(* IEC 61131-3 sources: PortalRobot/Portal_robot/Device/application/FB (part 2) *)

(* ---- FB_CELL_SAFETY.st ---- *)
FUNCTION_BLOCK FB_CELL_SAFETY
VAR_INPUT
	axDoorLockClosedInput : ARRAY [1..4] OF BOOL;
	axDoorUnlockButtonInput : ARRAY [1..4] OF BOOL;
	axMagazineMechanismBusy : ARRAY [1..2] OF BOOL; // Только новый механизм, включая фактическое движение оси
	axEmergencyStopButtonStationInput : ARRAY [1..4] OF BOOL;
	axEmergencyStopCabinetInput : ARRAY [1..2] OF BOOL;
	xEmergencyStopMpgInput : BOOL;
	xPhaseRelayOkInput    : BOOL;
	xPressureRelayOkInput : BOOL;
	xSafetyRelayOkInput   : BOOL;
	xCellStartButtonInput : BOOL;
	xCellStopButtonInput  : BOOL;
	xCellResetButtonInput : BOOL;
	xMpgAxisXInput : BOOL;
	xMpgAxisYInput : BOOL;
	xMpgAxisZInput : BOOL;
	xMpgMultiplier1Input : BOOL;
	xMpgMultiplier10Input : BOOL;
	xMpgMultiplier100Input : BOOL;
	xSafetyRelayReset : BOOL; // Импульс отдельного сброса реле безопасности
	astMagazineStatus : ARRAY [1..2] OF ST_MAGAZINE_STATUS;
	FaultRequest : ST_CELL_SAFETY_FAULT_REQUEST;
END_VAR
VAR_OUTPUT
	Status : ST_CELL_SAFETY_STATUS;
	Error  : ST_CELL_SAFETY_ERRORS;
	Diag   : ST_CELL_SAFETY_DIAG;
	FaultStatus : ST_FAULT_INJECTION_STATUS;
	astButtonStationIoStatus : ARRAY [1..4] OF ST_BUTTON_STATION_IO_STATUS;
	stFrontControlCabinetIoStatus : ST_CONTROL_CABINET_IO_STATUS;
	stRearControlCabinetIoStatus : ST_CONTROL_CABINET_IO_STATUS;
	stMpgIoStatus : ST_MPG_IO_STATUS;
	astEnclosureDoorStatus : ARRAY [1..4] OF ST_ENCLOSURE_DOOR_STATUS;
	axDoorUnlockOutput : ARRAY [1..4] OF BOOL;
	axDoorButtonLampOutput : ARRAY [1..4] OF BOOL;
	xSafetyRelayResetOutput : BOOL;
	xCellEnablePulse : BOOL;
	xCellDisablePulse : BOOL;
	xCellResetPulse : BOOL;
END_VAR
VAR
	fbFaultInjector : FB_CELL_SAFETY_FAULT_INJECTOR;
	axEmergencyStopStation : ARRAY [1..4] OF BOOL;
	axEmergencyStopCabinet : ARRAY [1..2] OF BOOL;
	axDoorLocked : ARRAY [1..4] OF BOOL;
	axDoorUnlockDemand : ARRAY [1..4] OF BOOL;
	axDoorSeenUnlocked : ARRAY [1..4] OF BOOL;
	artDoorButton : ARRAY [1..4] OF R_TRIG;
	rtSafetyRelayReset : R_TRIG;
	tpSafetyRelayReset : TP;
	rtCellStart : R_TRIG;
	rtCellStop : R_TRIG;
	rtCellReset : R_TRIG;
	xEmergencyStopMpg : BOOL;
	xPhaseRelayOk : BOOL;
	xPressureRelayOk : BOOL;
	xSafetyRelayOk : BOOL;
	dwLiveFaultMask : DWORD;
	uiDoor : UINT;
	uiMagazine : UINT;
END_VAR
VAR CONSTANT
	ERR_ESTOP_STATION_1 : DWORD := DWORD#16#0000_0001;
	ERR_ESTOP_STATION_2 : DWORD := DWORD#16#0000_0002;
	ERR_ESTOP_STATION_3 : DWORD := DWORD#16#0000_0004;
	ERR_ESTOP_STATION_4 : DWORD := DWORD#16#0000_0008;
	ERR_ESTOP_CABINET_FRONT : DWORD := DWORD#16#0000_0010;
	ERR_ESTOP_CABINET_REAR  : DWORD := DWORD#16#0000_0020;
	ERR_ESTOP_MPG      : DWORD := DWORD#16#0000_0040;
	ERR_PHASE_RELAY    : DWORD := DWORD#16#0000_0080;
	ERR_PRESSURE_RELAY : DWORD := DWORD#16#0000_0100;
	ERR_SAFETY_RELAY   : DWORD := DWORD#16#0000_0200;
	ERR_DOOR_1_UNLOCKED : DWORD := DWORD#16#0000_0400;
	ERR_DOOR_2_UNLOCKED : DWORD := DWORD#16#0000_0800;
	ERR_DOOR_3_UNLOCKED : DWORD := DWORD#16#0000_1000;
	ERR_DOOR_4_UNLOCKED : DWORD := DWORD#16#0000_2000;
	WRN_SAFETY_RESET_REJECTED : UINT := UINT#1;
	WRN_DOOR_1_UNLOCK_REJECTED : UINT := UINT#2;
END_VAR

// --- BEGIN IMPLEMENTATION ---

fbFaultInjector(Request := FaultRequest);
FaultStatus := fbFaultInjector.Status;

FOR uiDoor := UINT#1 TO UINT#4 DO
	axEmergencyStopStation[uiDoor] := axEmergencyStopButtonStationInput[uiDoor]
		OR fbFaultInjector.axEmergencyStopStation[uiDoor];
	axDoorLocked[uiDoor] := axDoorLockClosedInput[uiDoor]
		AND NOT fbFaultInjector.axDoorUnlocked[uiDoor];
	artDoorButton[uiDoor](CLK := axDoorUnlockButtonInput[uiDoor]);

	IF uiDoor <= UINT#2 THEN
		uiMagazine := UINT#1;
	ELSE
		uiMagazine := UINT#2;
	END_IF;
	astEnclosureDoorStatus[uiDoor].xUnlockAllowed := NOT astMagazineStatus[uiMagazine].xEnabled AND NOT axMagazineMechanismBusy[uiMagazine];
	axDoorButtonLampOutput[uiDoor] := astEnclosureDoorStatus[uiDoor].xUnlockAllowed;

	IF artDoorButton[uiDoor].Q THEN
		IF astEnclosureDoorStatus[uiDoor].xUnlockAllowed THEN
			axDoorUnlockDemand[uiDoor] := TRUE;
			axDoorSeenUnlocked[uiDoor] := FALSE;
		ELSE
			RaiseWarning(uiCode := WRN_DOOR_1_UNLOCK_REJECTED + uiDoor - UINT#1);
		END_IF;
	END_IF;

	// Команда держится до фактического цикла «замок открылся -> снова закрылся».
	// Если магазин включили поверх открытого доступа, выход снимается немедленно.
	IF NOT astEnclosureDoorStatus[uiDoor].xUnlockAllowed THEN
		axDoorUnlockDemand[uiDoor] := FALSE;
		axDoorSeenUnlocked[uiDoor] := FALSE;
	ELSIF axDoorUnlockDemand[uiDoor] THEN
		IF NOT axDoorLocked[uiDoor] THEN
			axDoorSeenUnlocked[uiDoor] := TRUE;
		ELSIF axDoorSeenUnlocked[uiDoor] THEN
			axDoorUnlockDemand[uiDoor] := FALSE;
			axDoorSeenUnlocked[uiDoor] := FALSE;
		END_IF;
	END_IF;

	axDoorUnlockOutput[uiDoor] := axDoorUnlockDemand[uiDoor];
	astEnclosureDoorStatus[uiDoor].xLocked := axDoorLocked[uiDoor];
	astEnclosureDoorStatus[uiDoor].xUnlockOutput := axDoorUnlockOutput[uiDoor];
	astButtonStationIoStatus[uiDoor].xEmergencyStopPressed := axEmergencyStopStation[uiDoor];
	astButtonStationIoStatus[uiDoor].xButtonPressed := axDoorUnlockButtonInput[uiDoor];
	astButtonStationIoStatus[uiDoor].xButtonLightOn := axDoorButtonLampOutput[uiDoor];
	Status.axEmergencyStopReleased[uiDoor] := NOT axEmergencyStopStation[uiDoor];
	Status.axDoorReady[uiDoor] := astEnclosureDoorStatus[uiDoor].xUnlockAllowed OR axDoorLocked[uiDoor];
	Status.axButtonStationPressed[uiDoor] := astButtonStationIoStatus[uiDoor].xButtonPressed;
	Status.axButtonStationLightOn[uiDoor] := astButtonStationIoStatus[uiDoor].xButtonLightOn;
END_FOR;

FOR uiDoor := UINT#1 TO UINT#2 DO
	axEmergencyStopCabinet[uiDoor] := axEmergencyStopCabinetInput[uiDoor]
		OR fbFaultInjector.axEmergencyStopCabinet[uiDoor];
	Status.axEmergencyStopReleased[uiDoor + UINT#4] := NOT axEmergencyStopCabinet[uiDoor];
END_FOR;
xEmergencyStopMpg := xEmergencyStopMpgInput OR fbFaultInjector.xEmergencyStopMpg;
Status.axEmergencyStopReleased[7] := NOT xEmergencyStopMpg;

xPhaseRelayOk := xPhaseRelayOkInput AND NOT fbFaultInjector.xPhaseRelayFault;
xPressureRelayOk := xPressureRelayOkInput AND NOT fbFaultInjector.xPressureRelayFault;
xSafetyRelayOk := xSafetyRelayOkInput AND NOT fbFaultInjector.xSafetyRelayFault;

rtSafetyRelayReset(CLK := xSafetyRelayReset);
Status.xSafetyRelayResetAllowed := NOT xSafetyRelayOk AND NOT tpSafetyRelayReset.Q;
IF rtSafetyRelayReset.Q AND NOT Status.xSafetyRelayResetAllowed THEN
	RaiseWarning(uiCode := WRN_SAFETY_RESET_REJECTED);
END_IF;
tpSafetyRelayReset(
	IN := rtSafetyRelayReset.Q AND Status.xSafetyRelayResetAllowed,
	PT := T#1S
);
// Разрешение проверяется на фронте команды; после запуска выдаём полный импульс 1 с.
xSafetyRelayResetOutput := tpSafetyRelayReset.Q;
Status.xSafetyRelayResetActive := xSafetyRelayResetOutput;

rtCellStart(CLK := xCellStartButtonInput);
rtCellStop(CLK := xCellStopButtonInput);
rtCellReset(CLK := xCellResetButtonInput);
xCellEnablePulse := rtCellStart.Q;
xCellDisablePulse := rtCellStop.Q;
xCellResetPulse := rtCellReset.Q;

stFrontControlCabinetIoStatus.xEmergencyStopPressed := axEmergencyStopCabinet[1];
stFrontControlCabinetIoStatus.xStartPressed := xCellStartButtonInput;
stFrontControlCabinetIoStatus.xStopPressed := xCellStopButtonInput;
stFrontControlCabinetIoStatus.xResetPressed := xCellResetButtonInput;
stRearControlCabinetIoStatus.xEmergencyStopPressed := axEmergencyStopCabinet[2];
stRearControlCabinetIoStatus.xStartPressed := FALSE;
stRearControlCabinetIoStatus.xStopPressed := FALSE;
stRearControlCabinetIoStatus.xResetPressed := FALSE;
stMpgIoStatus.xEmergencyStopPressed := xEmergencyStopMpg;
stMpgIoStatus.xAxisX := xMpgAxisXInput;
stMpgIoStatus.xAxisY := xMpgAxisYInput;
stMpgIoStatus.xAxisZ := xMpgAxisZInput;
stMpgIoStatus.xMultiplier1 := xMpgMultiplier1Input;
stMpgIoStatus.xMultiplier10 := xMpgMultiplier10Input;
stMpgIoStatus.xMultiplier100 := xMpgMultiplier100Input;

dwLiveFaultMask := DWORD#0;
IF axEmergencyStopStation[1] THEN dwLiveFaultMask := dwLiveFaultMask OR ERR_ESTOP_STATION_1; END_IF;
IF axEmergencyStopStation[2] THEN dwLiveFaultMask := dwLiveFaultMask OR ERR_ESTOP_STATION_2; END_IF;
IF axEmergencyStopStation[3] THEN dwLiveFaultMask := dwLiveFaultMask OR ERR_ESTOP_STATION_3; END_IF;
IF axEmergencyStopStation[4] THEN dwLiveFaultMask := dwLiveFaultMask OR ERR_ESTOP_STATION_4; END_IF;
IF axEmergencyStopCabinet[1] THEN dwLiveFaultMask := dwLiveFaultMask OR ERR_ESTOP_CABINET_FRONT; END_IF;
IF axEmergencyStopCabinet[2] THEN dwLiveFaultMask := dwLiveFaultMask OR ERR_ESTOP_CABINET_REAR; END_IF;
IF xEmergencyStopMpg THEN dwLiveFaultMask := dwLiveFaultMask OR ERR_ESTOP_MPG; END_IF;
IF NOT xPhaseRelayOk THEN dwLiveFaultMask := dwLiveFaultMask OR ERR_PHASE_RELAY; END_IF;
IF NOT xPressureRelayOk THEN dwLiveFaultMask := dwLiveFaultMask OR ERR_PRESSURE_RELAY; END_IF;
IF NOT xSafetyRelayOk THEN dwLiveFaultMask := dwLiveFaultMask OR ERR_SAFETY_RELAY; END_IF;
IF (astMagazineStatus[1].xEnabled OR axMagazineMechanismBusy[1]) AND NOT axDoorLocked[1] THEN dwLiveFaultMask := dwLiveFaultMask OR ERR_DOOR_1_UNLOCKED; END_IF;
IF (astMagazineStatus[1].xEnabled OR axMagazineMechanismBusy[1]) AND NOT axDoorLocked[2] THEN dwLiveFaultMask := dwLiveFaultMask OR ERR_DOOR_2_UNLOCKED; END_IF;
IF (astMagazineStatus[2].xEnabled OR axMagazineMechanismBusy[2]) AND NOT axDoorLocked[3] THEN dwLiveFaultMask := dwLiveFaultMask OR ERR_DOOR_3_UNLOCKED; END_IF;
IF (astMagazineStatus[2].xEnabled OR axMagazineMechanismBusy[2]) AND NOT axDoorLocked[4] THEN dwLiveFaultMask := dwLiveFaultMask OR ERR_DOOR_4_UNLOCKED; END_IF;

Error.dwErrorActive := dwLiveFaultMask;
Error.dwAlarmActive := dwLiveFaultMask;
IF dwLiveFaultMask <> DWORD#0 THEN
	Error.dwErrorLast := dwLiveFaultMask;
END_IF;
Status.xPhaseRelayOk := xPhaseRelayOk;
Status.xPressureRelayOk := xPressureRelayOk;
Status.xSafetyRelayOk := xSafetyRelayOk;
Status.xGlobalError := dwLiveFaultMask <> DWORD#0;
Status.xReady := NOT Status.xGlobalError;

(* ---- FB_GRIPPER_SIMULATION.st ---- *)
FUNCTION_BLOCK FB_GRIPPER_SIMULATION
VAR_INPUT
	Command : ST_GRIPPER_COMMAND; // Команда управления захватом

    xSimGripper1Fault : BOOL; // Имитация неисправности первого захвата
    xSimGripper2Fault : BOOL; // Имитация неисправности второго захвата
    xSimRotationFault : BOOL; // Имитация неисправности поворота
    xSimGlobalFault   : BOOL; // Имитация общей неисправности захвата

    tGripperTime : TIME := T#500MS; // Время открытия или закрытия захвата
    tRotateTime  : TIME := T#700MS; // Время поворота захвата
END_VAR
VAR_OUTPUT
	Status : ST_GRIPPER_STATUS; // Рабочие статусы захвата
	Diag   : ST_GRIPPER_DIAG; // Состояние автомата и активное действие
	Error  : ST_GRIPPER_ERRORS; // Активные и последние ошибки
END_VAR
VAR
	eState        : E_GRIPPER_STATE := E_GRIPPER_STATE.IDLE; // Текущее состояние автомата захвата
    eActiveAction : E_ROBOT_ACTION := E_ROBOT_ACTION.NONE; // Выполняемое действие захвата

    tonAction      : TON; // Таймер выполнения действия
    xActionFault   : BOOL; // Неисправность, относящаяся к текущему действию
	xActionValid   : BOOL; // Получено допустимое действие захвата
	xActionRequired: BOOL; // Для действия требуется физическое переключение
    tActionTime    : TIME; // Нормативное время текущего действия
    xInitialized   : BOOL; // Начальные состояния установлены
END_VAR
VAR CONSTANT
	ERR_GRIPPER_1   : DWORD := DWORD#16#0000_0001; // Ошибка первого захвата
    ERR_GRIPPER_2   : DWORD := DWORD#16#0000_0002; // Ошибка второго захвата
    ERR_GRIP_ROTATE : DWORD := DWORD#16#0000_0004; // Ошибка механизма поворота
    ERR_GRIP_ACTION : DWORD := DWORD#16#0000_0008; // Недопустимое действие захвата
    ERR_GRIP_GLOBAL : DWORD := DWORD#16#0000_0010; // Общая ошибка захвата
END_VAR

// --- BEGIN IMPLEMENTATION ---

IF NOT xInitialized THEN
    Status.xGripper1Open := TRUE;
    Status.xGripper1Closed := FALSE;

    Status.xGripper2Open := TRUE;
    Status.xGripper2Closed := FALSE;

    Status.xRotatedToBlank := TRUE;
    Status.xRotatedToDetail := FALSE;

    xInitialized := TRUE;
END_IF;

xActionFault := FALSE;
tActionTime := tGripperTime;

CASE eActiveAction OF

    E_ROBOT_ACTION.UNCLAMP_1,
    E_ROBOT_ACTION.CLAMP_1:
        xActionFault := xSimGripper1Fault;

    E_ROBOT_ACTION.UNCLAMP_2,
    E_ROBOT_ACTION.CLAMP_2:
        xActionFault := xSimGripper2Fault;

    E_ROBOT_ACTION.ROTATE_TO_BLANK,
    E_ROBOT_ACTION.ROTATE_TO_DETAIL:
        xActionFault := xSimRotationFault;
        tActionTime := tRotateTime;

END_CASE;

tonAction(
    IN := (eState = E_GRIPPER_STATE.EXECUTE)
          AND NOT xActionFault
          AND NOT xSimGlobalFault,
    PT := tActionTime
);

CASE eState OF

    E_GRIPPER_STATE.IDLE:

        Status.xBusy := FALSE;
        Status.xDone := FALSE;
        Status.xError := FALSE;

        IF Command.xExecute THEN
            eActiveAction := Command.eAction;
			xActionValid := TRUE;
			xActionRequired := TRUE;

            CASE Command.eAction OF

				E_ROBOT_ACTION.UNCLAMP_1:
					xActionRequired := NOT Status.xGripper1Open;

				E_ROBOT_ACTION.CLAMP_1:
					xActionRequired := NOT Status.xGripper1Closed;

				E_ROBOT_ACTION.UNCLAMP_2:
					xActionRequired := NOT Status.xGripper2Open;

				E_ROBOT_ACTION.CLAMP_2:
					xActionRequired := NOT Status.xGripper2Closed;

				E_ROBOT_ACTION.ROTATE_TO_BLANK:
					xActionRequired := NOT Status.xRotatedToBlank;

				E_ROBOT_ACTION.ROTATE_TO_DETAIL:
					xActionRequired := NOT Status.xRotatedToDetail;

            ELSE
				xActionValid := FALSE;
                Error.dwErrorActive := Error.dwErrorActive OR ERR_GRIP_ACTION;
                eState := E_GRIPPER_STATE.ERROR;
            END_CASE;

			IF xActionValid THEN
				IF xActionRequired THEN
					eState := E_GRIPPER_STATE.EXECUTE;
				ELSE
					eState := E_GRIPPER_STATE.DONE;
				END_IF;
			END_IF;
        END_IF;

    E_GRIPPER_STATE.EXECUTE:

        Status.xBusy := TRUE;
        Status.xDone := FALSE;

        IF xSimGlobalFault THEN
            Error.dwErrorActive := Error.dwErrorActive OR ERR_GRIP_GLOBAL;
            eState := E_GRIPPER_STATE.ERROR;

        ELSIF xActionFault THEN

            CASE eActiveAction OF

                E_ROBOT_ACTION.UNCLAMP_1,
                E_ROBOT_ACTION.CLAMP_1:
                    Error.dwErrorActive := Error.dwErrorActive OR ERR_GRIPPER_1;

                E_ROBOT_ACTION.UNCLAMP_2,
                E_ROBOT_ACTION.CLAMP_2:
                    Error.dwErrorActive := Error.dwErrorActive OR ERR_GRIPPER_2;

                E_ROBOT_ACTION.ROTATE_TO_BLANK,
                E_ROBOT_ACTION.ROTATE_TO_DETAIL:
                    Error.dwErrorActive := Error.dwErrorActive OR ERR_GRIP_ROTATE;

            END_CASE;

            eState := E_GRIPPER_STATE.ERROR;

        ELSIF tonAction.Q THEN

            CASE eActiveAction OF

                E_ROBOT_ACTION.UNCLAMP_1:
                    Status.xGripper1Open := TRUE;
                    Status.xGripper1Closed := FALSE;

                E_ROBOT_ACTION.CLAMP_1:
                    Status.xGripper1Open := FALSE;
                    Status.xGripper1Closed := TRUE;

                E_ROBOT_ACTION.UNCLAMP_2:
                    Status.xGripper2Open := TRUE;
                    Status.xGripper2Closed := FALSE;

                E_ROBOT_ACTION.CLAMP_2:
                    Status.xGripper2Open := FALSE;
                    Status.xGripper2Closed := TRUE;

                E_ROBOT_ACTION.ROTATE_TO_BLANK:
                    Status.xRotatedToBlank := TRUE;
                    Status.xRotatedToDetail := FALSE;

                E_ROBOT_ACTION.ROTATE_TO_DETAIL:
                    Status.xRotatedToBlank := FALSE;
                    Status.xRotatedToDetail := TRUE;

            END_CASE;

            eState := E_GRIPPER_STATE.DONE;
        END_IF;

    E_GRIPPER_STATE.DONE:

        Status.xBusy := FALSE;
        Status.xDone := TRUE;

        IF NOT Command.xExecute THEN
            Status.xDone := FALSE;
            eActiveAction := E_ROBOT_ACTION.NONE;
            eState := E_GRIPPER_STATE.IDLE;
        END_IF;

    E_GRIPPER_STATE.ERROR:

        Status.xBusy := FALSE;
        Status.xDone := FALSE;
        Status.xError := TRUE;

        IF Command.xReset
        AND NOT Command.xExecute
        AND NOT xSimGlobalFault
        AND NOT xSimGripper1Fault
		AND NOT xSimGripper2Fault
		AND NOT xSimRotationFault THEN

			Error.dwErrorLast := Error.dwErrorActive;
            Error.dwErrorActive := DWORD#0;
            Status.xError := FALSE;
            eActiveAction := E_ROBOT_ACTION.NONE;
            eState := E_GRIPPER_STATE.IDLE;
        END_IF;

END_CASE;

Diag.eState := eState;
Diag.eActiveAction := eActiveAction;

IF Error.dwErrorActive <> DWORD#0 THEN
	Error.dwErrorLast := Error.dwErrorActive;
END_IF;

Error.stErrorActive := UpdateErrorView(dwError := Error.dwErrorActive);
Error.stErrorLast := UpdateErrorView(dwError := Error.dwErrorLast);
Error.dwAlarmActive := Error.dwErrorActive;

(* ---- FB_MACHINE.st ---- *)
FUNCTION_BLOCK FB_MACHINE
VAR_INPUT
    xExecute          : BOOL; // Запуск разрешённой операции обслуживания
    xReset            : BOOL; // Сброс ошибки конкретного станка
    xResetGlobal      : BOOL; // Общий сброс ошибок ячейки
    xGlobalError      : BOOL; // Глобальная ошибка ячейки
    xHmiSetBlank	  : BOOL; // Ручное подтверждение загруженной заготовки
    xHmiSetDetail     : BOOL; // Ручное подтверждение загруженной детали
    xHmiEnable        : BOOL; // Импульс включения станка в работу
    xHmiDisable       : BOOL; // Импульс отключения станка от работы
    xHmiAcceptRunCNC  : BOOL; // Импульс подтверждения запуска цикла обработки на станке
    xHmiRejectRunCNC  : BOOL; // Импульс отклонения запуска цикла обработки на станке
    xHmiAcceptDoor    : BOOL; // Импульс подтверждения оператора закрытии двери
    xHmiRejectDoor    : BOOL; // Импульс отклонения оператора закрытии двери
    xUseHmiCycleTime  : BOOL; // TRUE: использовать время цикла, заданное с HMI
    tHmiCycleTime     : TIME; // Начальная или постоянная оценка времени цикла
    stChangeRecipe    : ARRAY [0..40] OF ST_MACHINE_RECIPE; // Рецепт смены детали
    stLoadRecipe      : ARRAY [0..40] OF ST_MACHINE_RECIPE; // Рецепт загрузки заготовки
    stUnloadRecipe    : ARRAY [0..40] OF ST_MACHINE_RECIPE; // Рецепт выгрузки детали
    stPoints          : ST_MACHINE_POINTS; // Имена рабочих точек станка
    stRobotStatus     : ST_ROBOT_STATUS; // Статусы робота
    stMachineStatus   : ST_MACHINE_IO_STATUS; // Состояние исполнительных механизмов станка
END_VAR
VAR_OUTPUT
    Command : ST_MACHINE_COMMAND; // Команды станку и роботу
    Status  : ST_MACHINE_PUBLIC; // Публичные статусы станка
    Diag    : ST_MACHINE_DIAG; // Состояние автомата и выбранная операция
    Error   : ST_MACHINE_ERRORS; // Активные и последние ошибки
END_VAR
VAR
    eState                  : E_MACHINE_STATE := E_MACHINE_STATE.DISABLED; // Текущее состояние автомата
    ePartState              : E_PART_STATE := E_PART_STATE.UNKNOWN; // Состояние детали в патроне
    ePartType               : E_PART_TYPE := E_PART_TYPE.UNKNOWN; // Тип детали в патроне
    uiIndex                 : UINT; // Индекс команды рецепта
    tofErrorDoor            : TOF; // Контроль закрытия двери при нахождении робота внутри
    rtExectue               : R_TRIG; // Фронт команды запуска
    rtEnabledMachine        : R_TRIG; // Фронт команды включения
    rtDisabledMachine       : R_TRIG; // Фронт команды отключения
    rtResetMachine          : R_TRIG; // Фронт локального сброса ошибки станка
    rtCycleDone             : R_TRIG; // Фронт завершения цикла станка
    rtCycleStarted          : R_TRIG; // Фронт фактического запуска обработки
    ftCycleStopped          : F_TRIG; // Спад фактического цикла обработки
    rtSetBlankLoaded        : R_TRIG; // Фронт ручного подтверждения заготовки
    rtSetDetailLoaded       : R_TRIG; // Фронт ручного подтверждения детали
    ftChuckClamped          : F_TRIG; // Спад закрытия кулачков
    tonCycleMeasure         : TON; // Измерение длительности автоматического цикла
    xOperatorRunningCNC     : BOOL; // Оператор запустил цикл обработки с панели оператора
    xOperatorClosingDoor    : BOOL; // Оператор запустил закрытие дверей
    xAutoCycleCommanded     : BOOL; // Цикл был запущен этим блоком
    xCycleMeasureActive     : BOOL; // Измеряется текущий автоматический цикл
    xCycleMeasureValid      : BOOL; // Текущее измерение можно сохранить
    xMeasuredTimeValid      : BOOL; // Получено корректное измеренное время
    tMeasuredCycle          : TIME; // Последнее корректное измеренное время
    tExpectedCycle          : TIME; // Ожидаемое время текущего цикла
    xRetreatStarted         : BOOL; // Начат отход робота от станка
    xRobotInsideMachine     : BOOL; // Робот находится внутри рабочей зоны
    xRobotDone              : BOOL; // Робот освобождён алгоритмом станка
    xServiceDoorCloseDemand : BOOL; // Внутренний запрос закрытия двери
    xServiceDoorOpenDemand  : BOOL; // Внутренний запрос открытия двери
    xAutoDoorOpenLatched    : BOOL; // Защёлка автоматического открытия двери
    xRobotActionDone        : BOOL; // Запрошенное действие захвата уже выполнено
    xDisableRequest         : BOOL; // Сохранённый запрос отключения после операции или обработки
    eGrantedOperation       : E_MACHINE_OPERATION; // Разрешённая операция обслуживания
    eActualOperation        : E_MACHINE_OPERATION; // Выполняемая операция обслуживания
    stRecipe                : ARRAY [0..40] OF ST_MACHINE_RECIPE; // Активный рецепт операции
END_VAR

VAR CONSTANT
    ERR_WRONG_OPERATION     : DWORD := 1;   	// Приводит к глоабльной ошибке
    ERR_WRONG_COMMAND       : DWORD := 2;   	// Приводит к глобальной ошибке
    ERR_ROBOT_MOTION        : DWORD := 4;   	// Приводит к глобальной ошибке (Другой блок не создаём новую ошибку)
    ERR_ROBOT_ACTION        : DWORD := 8;   	// Приводит к глобальной ошибке (Другой блок не создаём новую ошибку)
    ERR_DOOR_OPEN  			: DWORD := 16;  	// Не приводит к глобальной ошибке, уезжаем в другой станок
    ERR_DOOR_CLOSE 			: DWORD := 32;  	// Не приводит к глобальной ошибке, уезжаем в другой станок
    ERR_CHUCK_OPEN 			: DWORD := 64;  	// Приводит к глобальной ошибке
    ERR_CHUCK_CLOSE 		: DWORD := 128; 	// Приводит к глобальной ошибке
    ERR_CYCLE_START			: DWORD := 256;     // Не приводит к глобальной ошибке
    ERR_SAFETY_STOP         : DWORD := 512;		// Глобальная ошибка из вне (Другой блок не создаём новую ошибку)
    ERR_UNKNOWN_DETAIL      : DWORD := 1024;    // Приводит к глобальной ошибке
    ERR_MACHINE_ALARM       : DWORD := 2048;    // Приводит к глобальной ошибке
    ERR_INDEX               : DWORD := 4096;    // Приводит к глобальной ошибке
    ERR_DOOR_ROBOT          : DWORD := 8192;    // Приводит к глобальной ошибке
    ERR_MACHINE_IDLE        : DWORD := 16384;   // Не приводит к глобальной ошибке

    // Ошибки, требующие формирования глобальной аварии ячейки.
    MASK_CRITICAL_ERROR		: DWORD :=
                                ERR_WRONG_OPERATION OR
                                ERR_WRONG_COMMAND OR
                                ERR_CHUCK_OPEN OR
                                ERR_CHUCK_CLOSE OR
                                ERR_UNKNOWN_DETAIL OR
                                ERR_MACHINE_ALARM OR
                                ERR_INDEX OR
                                ERR_DOOR_ROBOT;

    // Некритические ошибки конкретного станка.
    MASK_ALARM_ERROR		: DWORD :=
                                ERR_DOOR_OPEN OR
                                ERR_DOOR_CLOSE OR
                                ERR_CYCLE_START OR
                                ERR_MACHINE_IDLE;

    // Ошибки, полученные от других блоков или общей логики ячейки.
    MASK_EXTERNAL_ERROR  	: DWORD :=
                                ERR_SAFETY_STOP OR
                                ERR_ROBOT_ACTION OR
                                ERR_ROBOT_MOTION;

    WRN_RESET_ALARM_ACTIVE : UINT := 1; // Сброс отклонён из-за физической аварии станка
    WRN_RESET_GLOBAL_ERROR : UINT := 2; // Сброс отклонён из-за глобальной ошибки
    WRN_RESET_EXECUTE      : UINT := 3; // Сброс отклонён во время операции обслуживания

END_VAR

// --- BEGIN IMPLEMENTATION ---

(*
    1. Добавить таймауты (использовать уже существующие ошибки)
*)

rtEnabledMachine (CLK :=xHmiEnable);
rtDisabledMachine (CLK :=xHmiDisable);
rtResetMachine(CLK := xReset);
rtCycleDone(CLK := stMachineStatus.xCycleDone);
rtCycleStarted(CLK := stMachineStatus.xCycleActive);
ftCycleStopped(CLK := stMachineStatus.xCycleActive);
rtSetBlankLoaded(CLK := xHmiSetBlank);
rtSetDetailLoaded(CLK := xHmiSetDetail);
ftChuckClamped(CLK := stMachineStatus.xChuckClamped);

// Локальный сброс формирует одно предупреждение с конкретной причиной отказа.
IF rtResetMachine.Q
AND (eState = E_MACHINE_STATE.ERROR) THEN
    IF stMachineStatus.xAlarm THEN
        Diag.stWarning.uiCode := WRN_RESET_ALARM_ACTIVE;
    ELSIF xGlobalError THEN
        Diag.stWarning.uiCode := WRN_RESET_GLOBAL_ERROR;
    ELSIF xExecute THEN
        Diag.stWarning.uiCode := WRN_RESET_EXECUTE;
    ELSE
        Diag.stWarning.uiCode := UINT#0;
    END_IF;

    IF Diag.stWarning.uiCode <> UINT#0 THEN
        Diag.stWarning.udiSequence := Diag.stWarning.udiSequence + UDINT#1;
        IF Diag.stWarning.udiSequence = UDINT#0 THEN
            Diag.stWarning.udiSequence := UDINT#1;
        END_IF;
    END_IF;
END_IF;

IF rtDisabledMachine.Q THEN
    xDisableRequest := TRUE;
END_IF;

// Измеряются только циклы, запущенные автоматикой этого блока.
IF rtCycleStarted.Q THEN
    xCycleMeasureActive := xAutoCycleCommanded;
    xCycleMeasureValid := xAutoCycleCommanded;
END_IF;

IF xCycleMeasureActive
AND (stMachineStatus.xAlarm
    OR xGlobalError
    OR (eState = E_MACHINE_STATE.ERROR)
    OR (eState = E_MACHINE_STATE.DISABLED)) THEN
    xCycleMeasureValid := FALSE;
END_IF;

IF ftCycleStopped.Q THEN
    IF xCycleMeasureActive
    AND xCycleMeasureValid
    AND (tonCycleMeasure.ET > T#0S) THEN
        tMeasuredCycle := tonCycleMeasure.ET;
        xMeasuredTimeValid := TRUE;
    END_IF;
    xCycleMeasureActive := FALSE;
    xCycleMeasureValid := FALSE;
    xAutoCycleCommanded := FALSE;
END_IF;

tonCycleMeasure(
    IN := stMachineStatus.xCycleActive,
    PT := T#24H
);

// В автоматическом режиме до первого измерения используется время с HMI.
IF xUseHmiCycleTime THEN
    tExpectedCycle := tHmiCycleTime;
ELSIF xMeasuredTimeValid THEN
    tExpectedCycle := tMeasuredCycle;
ELSE
    tExpectedCycle := tHmiCycleTime;
END_IF;

// Команды по умолчанию
Command.stIo.xOpenDoor := FALSE;
Command.stIo.xCloseDoor := FALSE;
Command.stIo.xClampChuck := FALSE;
Command.stIo.xUnclampChuck := FALSE;
Command.stIo.xStartCycle := FALSE;
Command.stIo.xReset := xReset OR xResetGlobal;

Command.stRobot.xExecute := FALSE;
Command.stRobot.xStop := FALSE;
Command.stRobot.eAction := E_ROBOT_ACTION.NONE;
xServiceDoorOpenDemand := FALSE;
xServiceDoorCloseDemand := FALSE;

IF stMachineStatus.xChuckClamped AND NOT stMachineStatus.xAlarm THEN
    ePartState := E_PART_STATE.LOADED;
ELSIF stMachineStatus.xChuckUnclamped AND NOT stMachineStatus.xAlarm THEN
    ePartState := E_PART_STATE.EMPTY;
ELSE
    ePartState := E_PART_STATE.UNKNOWN;
END_IF

// // Ручное подтверждение состояния детали
// IF (eState = E_MACHINE_STATE.IDLE)
// AND NOT stMachineStatus.xCycleActive THEN
//     IF rtSetPartLoaded.Q THEN
//         ePartState := E_PART_STATE.LOADED;
//     END_IF;
//
//     IF rtSetPartEmpty.Q THEN
//         ePartState := E_PART_STATE.EMPTY;
//     END_IF;
// END_IF;

// Автоматическое открытие после окончания обработки
IF rtCycleDone.Q
    AND NOT stMachineStatus.xAlarm
    AND NOT stMachineStatus.xCycleActive
    AND (eState = E_MACHINE_STATE.IDLE)
    AND NOT xGlobalError THEN
    ePartType := E_PART_TYPE.DETAIL;
    xAutoDoorOpenLatched := TRUE;
END_IF;

IF stMachineStatus.xDoorOpen THEN
    xAutoDoorOpenLatched := FALSE;
END_IF;

eGrantedOperation := E_MACHINE_OPERATION.NONE;

IF (ePartState = E_PART_STATE.EMPTY)
AND (ePartType = E_PART_TYPE.UNKNOWN)
AND stRobotStatus.xBlankAvailable  THEN
    eGrantedOperation := E_MACHINE_OPERATION.LOAD;

ELSIF (ePartState = E_PART_STATE.LOADED)
AND (ePartType = E_PART_TYPE.DETAIL) THEN
    IF stRobotStatus.xBlankAvailable THEN
        eGrantedOperation := E_MACHINE_OPERATION.CHANGE;
    ELSE
        eGrantedOperation := E_MACHINE_OPERATION.UNLOAD;
    END_IF;
ELSIF (ePartState = E_PART_STATE.UNKNOWN) THEN
    eGrantedOperation := E_MACHINE_OPERATION.NONE;
END_IF;

// Включение и отключение блока
IF xDisableRequest
AND (((eState = E_MACHINE_STATE.IDLE) AND NOT stMachineStatus.xCycleActive)
    OR (eState = E_MACHINE_STATE.OPERATOR_CHOICE_PART)
    OR (eState = E_MACHINE_STATE.OPERATOR_CHOICE_DOOR)
    OR (eState = E_MACHINE_STATE.OPERATOR_CHOICE_RUN)) THEN
    eState := E_MACHINE_STATE.DISABLED;
ELSIF rtEnabledMachine.Q AND eState = E_MACHINE_STATE.DISABLED AND NOT stMachineStatus.xAlarm THEN
    IF ePartState = E_PART_STATE.EMPTY THEN
        eState := E_MACHINE_STATE.IDLE;
    ELSIF ePartState = E_PART_STATE.LOADED THEN
        eState := E_MACHINE_STATE.OPERATOR_CHOICE_PART;
    END_IF;
ELSIF rtEnabledMachine.Q AND eState = E_MACHINE_STATE.DISABLED AND stMachineStatus.xAlarm THEN
    eState := E_MACHINE_STATE.ERROR;
END_IF;

IF xGlobalError
AND Status.xBusy THEN
    Error.dwErrorActive := Error.dwErrorActive OR ERR_SAFETY_STOP;
    eState := E_MACHINE_STATE.ERROR;
END_IF;

IF stMachineStatus.xAlarm AND (eState = E_MACHINE_STATE.IDLE) THEN
    Error.dwErrorActive := Error.dwErrorActive OR ERR_MACHINE_IDLE;
    eState := E_MACHINE_STATE.ERROR;
END_IF

IF ((eState = E_MACHINE_STATE.OPERATOR_CHOICE_PART) OR (eState = E_MACHINE_STATE.OPERATOR_CHOICE_DOOR) OR (eState = E_MACHINE_STATE.OPERATOR_CHOICE_RUN))
AND ftChuckClamped.Q THEN
    eState := E_MACHINE_STATE.DISABLED;
END_IF;

IF (eState = E_MACHINE_STATE.DISABLED) OR (eState = E_MACHINE_STATE.ERROR) THEN
    xOperatorRunningCNC := FALSE;
    xOperatorClosingDoor := FALSE;
    ePartType :=   E_PART_TYPE.UNKNOWN;
END_IF
//Останавливаем робота, если кто-то попытался закрыть дверь в станке в момент его работы
tofErrorDoor(
            PT:= T#100MS,
            IN:=stMachineStatus.xDoorOpen
);

xRobotInsideMachine := (eState = E_MACHINE_STATE.ROBOT_ACTION)
                        OR (eState = E_MACHINE_STATE.ROBOT_MOVE)
                        OR (eState = E_MACHINE_STATE.RELEASE_ROBOT_ACTION);

IF xRobotInsideMachine AND NOT tofErrorDoor.Q THEN
    Command.stRobot.xStop := TRUE;
    Error.dwErrorActive := Error.dwErrorActive OR ERR_DOOR_ROBOT;
    eState := E_MACHINE_STATE.ERROR;
END_IF

CASE eState OF
    E_MACHINE_STATE.DISABLED:
        xDisableRequest := FALSE;
        IF NOT stMachineStatus.xCycleActive THEN
            xAutoCycleCommanded := FALSE;
        END_IF;

    E_MACHINE_STATE.OPERATOR_CHOICE_PART:
        IF rtSetDetailLoaded.Q AND NOT stMachineStatus.xAlarm THEN
            eState := E_MACHINE_STATE.IDLE;
            ePartType := E_PART_TYPE.DETAIL;
        ELSIF rtSetBlankLoaded.Q AND NOT stMachineStatus.xAlarm THEN
            eState := E_MACHINE_STATE.OPERATOR_CHOICE_DOOR;
            ePartType := E_PART_TYPE.PART;
        ELSIF stMachineStatus.xAlarm THEN
            Error.dwErrorActive := Error.dwErrorActive OR ERR_MACHINE_ALARM;
            eState := E_MACHINE_STATE.ERROR;
        END_IF;

    E_MACHINE_STATE.OPERATOR_CHOICE_DOOR:
        IF stMachineStatus.xDoorClosed
        AND NOT stMachineStatus.xAlarm THEN
            eState := E_MACHINE_STATE.OPERATOR_CHOICE_RUN;
        ELSIF NOT stMachineStatus.xDoorClosed
        AND xHmiAcceptDoor
        AND NOT stMachineStatus.xAlarm THEN
            xOperatorClosingDoor := TRUE;
            eState := E_MACHINE_STATE.DOOR_CLOSE;
        ELSIF NOT stMachineStatus.xDoorClosed
        AND xHmiRejectDoor
        AND NOT stMachineStatus.xAlarm THEN
            eState := E_MACHINE_STATE.DISABLED;
        ELSIF stMachineStatus.xAlarm THEN
            Error.dwErrorActive := Error.dwErrorActive OR ERR_MACHINE_ALARM;
            eState := E_MACHINE_STATE.ERROR;
        END_IF;

    E_MACHINE_STATE.OPERATOR_CHOICE_RUN:
        IF xHmiAcceptRunCNC AND NOT stMachineStatus.xAlarm THEN
            xOperatorRunningCNC := TRUE;
            eState := E_MACHINE_STATE.CYCLE_START;
        ELSIF xHmiRejectRunCNC AND NOT stMachineStatus.xAlarm THEN
            eState := E_MACHINE_STATE.DISABLED;
        ELSIF stMachineStatus.xAlarm THEN
            Error.dwErrorActive := Error.dwErrorActive OR ERR_MACHINE_ALARM;
            eState := E_MACHINE_STATE.ERROR;
        END_IF;

    E_MACHINE_STATE.IDLE:
        uiIndex := 0;
        xRobotDone := FALSE;
        IF xExecute THEN
            IF (stRobotStatus.eCurrentPoint = stPoints.eAbove)
            AND ePartState <> E_PART_STATE.UNKNOWN
            AND NOT stMachineStatus.xAlarm
            AND NOT stMachineStatus.xCycleActive
            AND NOT stRobotStatus.xBusy
            AND NOT stRobotStatus.xError
            AND NOT xGlobalError THEN
                eActualOperation := eGrantedOperation;
                eState := E_MACHINE_STATE.CHOSE;
            ELSIF ePartState = E_PART_STATE.UNKNOWN THEN
                Error.dwErrorActive := Error.dwErrorActive OR ERR_UNKNOWN_DETAIL;
                eState := E_MACHINE_STATE.ERROR ;
            END_IF
        END_IF

    E_MACHINE_STATE.CHOSE:
        CASE eActualOperation OF
            E_MACHINE_OPERATION.CHANGE:
                stRecipe := stChangeRecipe;
                eState := E_MACHINE_STATE.READ;
            E_MACHINE_OPERATION.LOAD:
                stRecipe := stLoadRecipe;
                eState := E_MACHINE_STATE.READ;
            E_MACHINE_OPERATION.UNLOAD:
                stRecipe := stUnloadRecipe;
                eState := E_MACHINE_STATE.READ;
        ELSE
            Error.dwErrorActive := Error.dwErrorActive OR ERR_WRONG_OPERATION ;
            eState := E_MACHINE_STATE.ERROR;
        END_CASE

    E_MACHINE_STATE.READ:
        CASE stRecipe[uiIndex].eCommand OF
            E_MACHINE_STATE.ROBOT_MOVE:
                eState := E_MACHINE_STATE.ROBOT_MOVE;

            E_MACHINE_STATE.ROBOT_ACTION:
                eState := E_MACHINE_STATE.ROBOT_ACTION;

            E_MACHINE_STATE.DOOR_OPEN:
                eState := E_MACHINE_STATE.DOOR_OPEN;

            E_MACHINE_STATE.DOOR_CLOSE:
                eState := E_MACHINE_STATE.DOOR_CLOSE;

            E_MACHINE_STATE.CHUCK_OPEN:
                eState := E_MACHINE_STATE.CHUCK_OPEN;

            E_MACHINE_STATE.CHUCK_CLOSE:
                eState := E_MACHINE_STATE.CHUCK_CLOSE;

            E_MACHINE_STATE.CYCLE_START:
                eState := E_MACHINE_STATE.CYCLE_START;

            E_MACHINE_STATE.DONE:
                eState := E_MACHINE_STATE.DONE;

        ELSE
            Error.dwErrorActive := Error.dwErrorActive OR ERR_WRONG_COMMAND;
            eState := E_MACHINE_STATE.ERROR;
        END_CASE

    E_MACHINE_STATE.NEXT:
            uiIndex := uiIndex + 1;
            IF uiIndex > 40 THEN
                Error.dwErrorActive := Error.dwErrorActive OR ERR_INDEX;
                eState := E_MACHINE_STATE.ERROR;
            ELSE
                eState := E_MACHINE_STATE.READ;
            END_IF;

    E_MACHINE_STATE.ROBOT_MOVE:
        Command.stRobot.xExecute  := TRUE;
        Command.stRobot.eAction   := E_ROBOT_ACTION.MOVE_TO_POINT;
        xRetreatStarted          := stRecipe[uiIndex].xRetreatStarted;
        IF stRecipe[uiIndex].stPoint = E_MACHINE_POINTS.ABOVE  THEN
            Command.stRobot.eSetPoint := stPoints.eAbove;
        ELSIF stRecipe[uiIndex].stPoint = E_MACHINE_POINTS.CHUCK THEN
            Command.stRobot.eSetPoint := stPoints.eChuck;
        ELSIF stRecipe[uiIndex].stPoint = E_MACHINE_POINTS.CHUCK_APPROACH THEN
            Command.stRobot.eSetPoint := stPoints.eChuckApproach;
        ELSIF stRecipe[uiIndex].stPoint = E_MACHINE_POINTS.INSIDE THEN
            Command.stRobot.eSetPoint := stPoints.eInside;
        END_IF

        IF stRobotStatus.xError THEN
            Error.dwErrorActive := Error.dwErrorActive OR ERR_ROBOT_MOTION;
            eState := E_MACHINE_STATE.ERROR ;

        ELSIF stMachineStatus.xAlarm THEN
            Command.stRobot.xStop := TRUE;
            Error.dwErrorActive := Error.dwErrorActive OR ERR_MACHINE_ALARM;
            eState := E_MACHINE_STATE.ERROR ;

        ELSIF stRobotStatus.xDone THEN
            eState := E_MACHINE_STATE.RELEASE_ROBOT_ACTION;

        END_IF;

    E_MACHINE_STATE.ROBOT_ACTION:
        xRobotActionDone := FALSE;

        CASE stRecipe[uiIndex].eRobotAction OF
            E_ROBOT_ACTION.UNCLAMP_1:
                xRobotActionDone := stRobotStatus.xGripper1Open;
            E_ROBOT_ACTION.CLAMP_1:
                xRobotActionDone := stRobotStatus.xGripper1Closed;
            E_ROBOT_ACTION.UNCLAMP_2:
                xRobotActionDone := stRobotStatus.xGripper2Open;
            E_ROBOT_ACTION.CLAMP_2:
                xRobotActionDone := stRobotStatus.xGripper2Closed;
            E_ROBOT_ACTION.ROTATE_TO_BLANK:
                xRobotActionDone := stRobotStatus.xRotatedToBlank;
            E_ROBOT_ACTION.ROTATE_TO_DETAIL:
                xRobotActionDone := stRobotStatus.xRotatedToDetail;
        END_CASE;

        IF xRobotActionDone THEN
            eState := E_MACHINE_STATE.NEXT;
        ELSE
            Command.stRobot.xExecute := TRUE;
            Command.stRobot.eAction := stRecipe[uiIndex].eRobotAction;
        END_IF;

        IF (eState = E_MACHINE_STATE.ROBOT_ACTION)
        AND stMachineStatus.xAlarm THEN
            Command.stRobot.xStop := TRUE;
            Error.dwErrorActive := Error.dwErrorActive OR ERR_MACHINE_ALARM;
            eState := E_MACHINE_STATE.ERROR ;

        ELSIF (eState = E_MACHINE_STATE.ROBOT_ACTION)
        AND stRobotStatus.xError THEN
            Error.dwErrorActive := Error.dwErrorActive OR ERR_ROBOT_ACTION;
            eState := E_MACHINE_STATE.ERROR ;

        ELSIF (eState = E_MACHINE_STATE.ROBOT_ACTION)
        AND stRobotStatus.xDone THEN
            eState := E_MACHINE_STATE.RELEASE_ROBOT_ACTION;
        END_IF;

    E_MACHINE_STATE.RELEASE_ROBOT_ACTION:
        IF NOT stRobotStatus.xBusy
        AND NOT stRobotStatus.xDone
        AND NOT stRobotStatus.xError THEN
            xRobotDone := stRecipe[uiIndex].xRobotDone;
            eState := E_MACHINE_STATE.NEXT;

        ELSIF stRobotStatus.xError AND  stRecipe[uiIndex].eRobotAction = E_ROBOT_ACTION.MOVE_TO_POINT THEN
            Error.dwErrorActive := Error.dwErrorActive OR ERR_ROBOT_MOTION;
            eState := E_MACHINE_STATE.ERROR;

        ELSIF stRobotStatus.xError THEN
            Error.dwErrorActive := Error.dwErrorActive OR ERR_ROBOT_ACTION;
            eState := E_MACHINE_STATE.ERROR;
        END_IF;

    E_MACHINE_STATE.DOOR_OPEN:
        xServiceDoorOpenDemand := TRUE;

        IF stMachineStatus.xDoorOpen
        AND NOT stMachineStatus.xAlarm THEN
            xServiceDoorOpenDemand := FALSE;
            eState := E_MACHINE_STATE.NEXT;
        ELSIF stMachineStatus.xAlarm THEN
            Error.dwErrorActive := Error.dwErrorActive OR ERR_DOOR_OPEN;
            eState := E_MACHINE_STATE.ERROR;
        END_IF;

    E_MACHINE_STATE.DOOR_CLOSE:
        xServiceDoorCloseDemand := TRUE;

        IF stMachineStatus.xDoorClosed
        AND NOT stMachineStatus.xAlarm THEN
            xServiceDoorCloseDemand := FALSE;
            IF NOT xOperatorClosingDoor THEN
                eState := E_MACHINE_STATE.NEXT;
            ELSIF xOperatorClosingDoor THEN
                eState := E_MACHINE_STATE.OPERATOR_CHOICE_RUN;
                xOperatorClosingDoor := FALSE;
            END_IF;
        ELSIF stMachineStatus.xAlarm THEN
            Error.dwErrorActive := Error.dwErrorActive OR ERR_DOOR_CLOSE;
            eState := E_MACHINE_STATE.ERROR;
        END_IF;

    E_MACHINE_STATE.CHUCK_OPEN:
        Command.stIo.xUnclampChuck := TRUE;

        IF stMachineStatus.xChuckUnclamped
        AND NOT stMachineStatus.xAlarm  THEN
            Command.stIo.xUnclampChuck := FALSE;
            ePartType := E_PART_TYPE.UNKNOWN;
               eState := E_MACHINE_STATE.NEXT;
        ELSIF stMachineStatus.xAlarm THEN
            Command.stIo.xUnclampChuck := FALSE;
            Error.dwErrorActive := Error.dwErrorActive OR ERR_CHUCK_OPEN;
            eState := E_MACHINE_STATE.ERROR;
        END_IF;

    E_MACHINE_STATE.CHUCK_CLOSE:
        Command.stIo.xClampChuck := TRUE;

        IF stMachineStatus.xChuckClamped
        AND NOT stMachineStatus.xAlarm  THEN
            Command.stIo.xClampChuck := FALSE;
            ePartType := E_PART_TYPE.PART;
               eState := E_MACHINE_STATE.NEXT;
        ELSIF stMachineStatus.xAlarm THEN
            Command.stIo.xClampChuck := FALSE;
            Error.dwErrorActive := Error.dwErrorActive OR ERR_CHUCK_CLOSE;
            eState := E_MACHINE_STATE.ERROR;
        END_IF;

    E_MACHINE_STATE.CYCLE_START:
        IF stMachineStatus.xChuckClamped
        AND stMachineStatus.xDoorClosed THEN
            Command.stIo.xStartCycle := TRUE;
            xAutoCycleCommanded := TRUE;
        END_IF;

        IF stMachineStatus.xCycleActive AND NOT stMachineStatus.xAlarm THEN
            Command.stIo.xStartCycle := FALSE;
            IF NOT xOperatorRunningCNC THEN
                eState := E_MACHINE_STATE.NEXT;
            ELSIF xOperatorRunningCNC THEN
                xOperatorRunningCNC := FALSE;
                eState := E_MACHINE_STATE.IDLE;
            END_IF;
        ELSIF stMachineStatus.xAlarm THEN
            Command.stIo.xStartCycle := FALSE;
            Error.dwErrorActive := Error.dwErrorActive OR ERR_CYCLE_START;
            eState := E_MACHINE_STATE.ERROR;
        END_IF;

    E_MACHINE_STATE.DONE:
        CASE eActualOperation OF
            E_MACHINE_OPERATION.CHANGE, E_MACHINE_OPERATION.LOAD:
                eActualOperation := E_MACHINE_OPERATION.NONE;
                ePartState := E_PART_STATE.LOADED;
            E_MACHINE_OPERATION.UNLOAD:
                eActualOperation := E_MACHINE_OPERATION.NONE;
                ePartState := E_PART_STATE.EMPTY;
        END_CASE

        IF NOT xExecute THEN
            xRobotDone := FALSE;
            eState := E_MACHINE_STATE.IDLE;
        END_IF

    E_MACHINE_STATE.ERROR:
        uiIndex := 0;
        eActualOperation := E_MACHINE_OPERATION.NONE;
        eGrantedOperation := E_MACHINE_OPERATION.NONE;
        IF NOT stMachineStatus.xCycleActive THEN
            xAutoCycleCommanded := FALSE;
        END_IF;

        IF (xReset OR xResetGlobal)
        AND NOT xGlobalError
        AND NOT xExecute
        AND NOT stMachineStatus.xAlarm THEN
            Error.dwErrorLast := Error.dwErrorActive;
            Error.dwErrorActive := DWORD#0;
            eState := E_MACHINE_STATE.DISABLED;
        END_IF;
END_CASE;

IF (eState <> E_MACHINE_STATE.ERROR)
AND NOT xGlobalError THEN
    IF xServiceDoorCloseDemand
    AND NOT (xAutoDoorOpenLatched OR xServiceDoorOpenDemand)
    AND NOT stMachineStatus.xAlarm THEN
        Command.stIo.xCloseDoor := TRUE;

    ELSIF (xAutoDoorOpenLatched OR xServiceDoorOpenDemand)
    AND NOT xServiceDoorCloseDemand
    AND NOT stMachineStatus.xCycleActive
    AND NOT stMachineStatus.xAlarm THEN
        Command.stIo.xOpenDoor := TRUE;
    END_IF;
END_IF;

Status.xCanAcceptService := (eState = E_MACHINE_STATE.IDLE)
            AND ePartState <> E_PART_STATE.UNKNOWN
            AND NOT stMachineStatus.xAlarm
            AND NOT stMachineStatus.xCycleActive
            AND NOT xGlobalError;

Status.xEnabled := eState <> E_MACHINE_STATE.DISABLED;
Status.xDisablePending := xDisableRequest AND Status.xEnabled;
Status.xProcessing := stMachineStatus.xCycleActive;
Status.xPartReady := stMachineStatus.xCycleDone;
Status.xServiceRequired := (eGrantedOperation <> E_MACHINE_OPERATION.NONE)
    AND (eState = E_MACHINE_STATE.IDLE);
Status.xRobotReleased := xRobotDone;
Status.xDone := (eState = E_MACHINE_STATE.DONE);
Status.xBusy :=  (eState <> E_MACHINE_STATE.IDLE)
                AND (eState <> E_MACHINE_STATE.DISABLED)
                AND (eState <> E_MACHINE_STATE.ERROR)
                AND (eState <> E_MACHINE_STATE.DONE)
                AND (eState <> E_MACHINE_STATE.OPERATOR_CHOICE_PART)
                AND (eState <> E_MACHINE_STATE.OPERATOR_CHOICE_RUN)
                AND (eState <> E_MACHINE_STATE.OPERATOR_CHOICE_DOOR)
                AND NOT ((eState = E_MACHINE_STATE.CYCLE_START) AND xOperatorRunningCNC)
                AND NOT ((eState = E_MACHINE_STATE.DOOR_CLOSE) AND xOperatorClosingDoor);
Status.xError := (eState = E_MACHINE_STATE.ERROR);
Status.xCriticalError := (Error.dwErrorActive AND MASK_CRITICAL_ERROR) <> DWORD#0;
Status.xAlarmError    := (Error.dwErrorActive AND MASK_ALARM_ERROR) <> DWORD#0;
Status.xExternalError := (Error.dwErrorActive AND MASK_EXTERNAL_ERROR) <> DWORD#0;
Error.dwAlarmActive := Error.dwErrorActive AND NOT MASK_EXTERNAL_ERROR;
Status.xDoorOpen := stMachineStatus.xDoorOpen;
Status.xAlarm := stMachineStatus.xAlarm;
Status.eRecommendedOperation := eGrantedOperation;
Status.ePartState := ePartState;
Status.ePartType := ePartType;
Status.eAbovePoint := stPoints.eAbove;
Status.tCycleExpected := tExpectedCycle;
Status.tCycleElapsed := tonCycleMeasure.ET;
Status.tMeasuredCycle := tMeasuredCycle;
Status.xCycleTimeValid := tExpectedCycle > T#0S;
Status.xMeasuredTimeValid := xMeasuredTimeValid;
Status.xCycleOvertime := FALSE;
Status.tRemaining := T#0S;

IF stMachineStatus.xCycleActive
AND Status.xCycleTimeValid THEN
    IF Status.tCycleElapsed < Status.tCycleExpected THEN
        Status.tRemaining := Status.tCycleExpected - Status.tCycleElapsed;
    ELSE
        Status.xCycleOvertime := TRUE;
    END_IF;
END_IF;

Diag.eState := eState;
Diag.eGrantedOperation := eGrantedOperation;
Diag.eActualOperation := eActualOperation;

IF Error.dwErrorActive <> DWORD#0 THEN
    Error.dwErrorLast := Error.dwErrorActive;
END_IF;

Error.stErrorActive := UpdateErrorView(dwError := Error.dwErrorActive);
Error.stErrorLast := UpdateErrorView(dwError := Error.dwErrorLast);

(* ---- FB_MACHINE_SIMULATION.st ---- *)
FUNCTION_BLOCK FB_MACHINE_SIMULATION
VAR_INPUT
    Command : ST_MACHINE_IO_COMMAND; // Команды исполнительным механизмам

    xSimMachineAlarm : BOOL; // Имитация общей аварии станка
    xSimDoorFault    : BOOL; // Имитация неисправности двери
    xSimChuckFault   : BOOL; // Имитация неисправности патрона

    tDoorTime  : TIME := T#1S; // Время открытия или закрытия двери
    tChuckTime : TIME := T#1S; // Время зажима или разжима патрона
    tCycleTime : TIME := T#47S; // Время цикла обработки
END_VAR

VAR_OUTPUT
    Status : ST_MACHINE_IO_STATUS; // Состояние исполнительных механизмов
	Diag   : ST_MACHINE_SIM_DIAG; // Текущие действия симулятора
	Error  : ST_MACHINE_SIM_ERRORS; // Активные и последние ошибки
END_VAR
VAR CONSTANT
	ERR_MACHINE_ALARM : DWORD := DWORD#16#0000_0001; // Авария станка
	ERR_DOOR_FAULT    : DWORD := DWORD#16#0000_0002; // Ошибка двери
	ERR_CHUCK_FAULT   : DWORD := DWORD#16#0000_0004; // Ошибка патрона
END_VAR

VAR
    rtStartCycle : R_TRIG; // Фронт команды запуска цикла

    tonDoorOpen   : TON; // Таймер открытия двери
    tonDoorClose  : TON; // Таймер закрытия двери
    tonChuckClamp : TON; // Таймер зажима патрона
    tonChuckOpen  : TON; // Таймер разжима патрона
    tonCycleStart : TON; // Таймер подтверждения запуска цикла
    tonCycle      : TON; // Таймер обработки

    xDoorOpening   : BOOL; // Выполняется открытие двери
    xDoorClosing   : BOOL; // Выполняется закрытие двери
    xChuckClamping : BOOL; // Выполняется зажим патрона
    xChuckOpening  : BOOL; // Выполняется разжим патрона
    xCycleStarting : BOOL; // Выполняется запуск цикла

    xAlarmLatched : BOOL; // Защёлкнутая авария симулятора
    xInitialized  : BOOL; // Начальные состояния установлены
END_VAR

// --- BEGIN IMPLEMENTATION ---

// =====================================================
// Первичная инициализация
// =====================================================

IF NOT xInitialized THEN
    Status.xDoorOpen := FALSE;
    Status.xDoorClosed := TRUE;

    Status.xChuckClamped := TRUE;
    Status.xChuckUnclamped := FALSE;

    Status.xCycleActive := FALSE;
    Status.xCycleDone := FALSE;
    Status.xAlarm := FALSE;

    xInitialized := TRUE;
END_IF;

// =====================================================
// Детектор запуска цикла
// =====================================================

rtStartCycle(CLK := Command.xStartCycle);

// =====================================================
// Формирование и сброс аварии
// =====================================================

IF xSimMachineAlarm THEN
	Error.dwErrorActive := Error.dwErrorActive OR ERR_MACHINE_ALARM;
END_IF;

IF xSimDoorFault
AND (xDoorOpening OR xDoorClosing) THEN
	Error.dwErrorActive := Error.dwErrorActive OR ERR_DOOR_FAULT;
END_IF;

IF xSimChuckFault
AND (xChuckClamping OR xChuckOpening) THEN
	Error.dwErrorActive := Error.dwErrorActive OR ERR_CHUCK_FAULT;
END_IF;

IF Command.xReset
AND NOT xSimMachineAlarm
AND NOT xSimDoorFault
AND NOT xSimChuckFault THEN
	Error.dwErrorLast := Error.dwErrorActive;
	Error.dwErrorActive := DWORD#0;
END_IF;

xAlarmLatched := Error.dwErrorActive <> DWORD#0;

// =====================================================
// Приём команд станка
// =====================================================

IF NOT xAlarmLatched THEN

    // Открытие двери
    IF Command.xOpenDoor
    AND NOT Status.xDoorOpen
    AND NOT Status.xCycleActive THEN
        xDoorOpening := TRUE;
        xDoorClosing := FALSE;
    END_IF;

    // Закрытие двери
    IF Command.xCloseDoor
    AND NOT Status.xDoorClosed THEN
        xDoorClosing := TRUE;
        xDoorOpening := FALSE;
    END_IF;

    // Зажим патрона
    IF Command.xClampChuck
    AND NOT Status.xChuckClamped
    AND NOT Status.xCycleActive THEN
        xChuckClamping := TRUE;
        xChuckOpening := FALSE;
    END_IF;

    // Разжим патрона
    IF Command.xUnclampChuck
    AND NOT Status.xChuckUnclamped
    AND NOT Status.xCycleActive THEN
        xChuckOpening := TRUE;
        xChuckClamping := FALSE;
    END_IF;

    // Запуск обработки
    IF rtStartCycle.Q
    AND Status.xDoorClosed
    AND Status.xChuckClamped
    AND NOT Status.xCycleActive THEN
        xCycleStarting := TRUE;
        Status.xCycleDone := FALSE;
    END_IF;

END_IF;

// =====================================================
// Таймеры механизмов
// =====================================================

tonDoorOpen(
    IN := xDoorOpening AND NOT xSimDoorFault,
    PT := tDoorTime
);

tonDoorClose(
    IN := xDoorClosing AND NOT xSimDoorFault,
    PT := tDoorTime
);

tonChuckClamp(
    IN := xChuckClamping AND NOT xSimChuckFault,
    PT := tChuckTime
);

tonChuckOpen(
    IN := xChuckOpening AND NOT xSimChuckFault,
    PT := tChuckTime
);

tonCycleStart(
    IN := xCycleStarting,
    PT := T#200MS
);

tonCycle(
    IN := Status.xCycleActive AND NOT xAlarmLatched,
    PT := tCycleTime
);

// =====================================================
// Завершение открытия двери
// =====================================================

IF tonDoorOpen.Q THEN
    Status.xDoorOpen := TRUE;
    Status.xDoorClosed := FALSE;

    xDoorOpening := FALSE;
END_IF;

// =====================================================
// Завершение закрытия двери
// =====================================================

IF tonDoorClose.Q THEN
    Status.xDoorClosed := TRUE;
    Status.xDoorOpen := FALSE;

    xDoorClosing := FALSE;
END_IF;

// =====================================================
// Завершение зажима патрона
// =====================================================

IF tonChuckClamp.Q THEN
    Status.xChuckClamped := TRUE;
    Status.xChuckUnclamped := FALSE;

    xChuckClamping := FALSE;
END_IF;

// =====================================================
// Завершение разжима патрона
// =====================================================

IF tonChuckOpen.Q THEN
    Status.xChuckUnclamped := TRUE;
    Status.xChuckClamped := FALSE;

    xChuckOpening := FALSE;
END_IF;

// =====================================================
// Запуск цикла
// =====================================================

IF tonCycleStart.Q THEN
    Status.xCycleActive := TRUE;
    xCycleStarting := FALSE;
END_IF;

// =====================================================
// Завершение цикла
// =====================================================

IF tonCycle.Q THEN
    Status.xCycleActive := FALSE;
    Status.xCycleDone := TRUE;
END_IF;

// =====================================================
// Реакция на аварийное состояние
// =====================================================

IF xAlarmLatched THEN
    Status.xCycleActive := FALSE;

    xDoorOpening := FALSE;
    xDoorClosing := FALSE;

    xChuckClamping := FALSE;
    xChuckOpening := FALSE;

    xCycleStarting := FALSE;
END_IF;

// =====================================================
// Выходной статус
// =====================================================

Status.xAlarm := xAlarmLatched;
Status.xReady := NOT xAlarmLatched AND NOT Status.xCycleActive;

Diag.xDoorOpening := xDoorOpening;
Diag.xDoorClosing := xDoorClosing;
Diag.xChuckClamping := xChuckClamping;
Diag.xChuckOpening := xChuckOpening;
Diag.xCycleStarting := xCycleStarting;

IF Error.dwErrorActive <> DWORD#0 THEN
	Error.dwErrorLast := Error.dwErrorActive;
END_IF;

Error.stErrorActive := UpdateErrorView(dwError := Error.dwErrorActive);
Error.stErrorLast := UpdateErrorView(dwError := Error.dwErrorLast);

(* ---- FB_MAGAZINE.st ---- *)
FUNCTION_BLOCK FB_MAGAZINE
VAR_INPUT
	stRobotStatus     : ST_ROBOT_STATUS; // Текущие статусы робота
	stMagazineCommand : ST_MAGAZINE_COMMAND; // Команда магазина от автоматической логики
	stHmiCommand      : ST_ROBOT_COMMAND; // Ручная команда магазина с HMI
	xManual           : BOOL; // Разрешение ручного управления
	xReset            : BOOL; // Сброс ошибок магазина
	xGlobalError      : BOOL; // Глобальная ошибка ячейки
	xMode             : BOOL; // Режим робота: TRUE — Modbus, FALSE — SoftMotion
	xHmiEnable        : BOOL; // Импульс включения магазина с HMI
	xHmiDisable       : BOOL; // Импульс отключения магазина с HMI
	xHmiFillBlanks    : BOOL; // Заполнить все активные слоты матрицы заготовками
	xHmiClear         : BOOL; // Полностью очистить содержимое магазина
	xHmiCycleSlot     : BOOL; // Переключить содержимое выбранного слота
	uiHmiEditSlot     : UINT; // Номер слота для ручного редактирования
	uiRows            : UINT; // Число строк матрицы магазина
	uiColumns         : UINT; // Число столбцов матрицы магазина
	lrPitchX          : LREAL; // Шаг между слотами по оси X
	lrPitchY          : LREAL; // Шаг между слотами по оси Y
	lrSafeZ_1           : LREAL; // Безопасная координата по оси Z
	lrSafeZ_2     : LREAL; // Безопасная координата по оси Z (при смене детали на заготовку)
END_VAR
VAR_OUTPUT
	Command : ST_ROBOT_COMMAND; // Текущая пошаговая команда роботу
	Status  : ST_MAGAZINE_STATUS; // Рабочие статусы магазина
	Diag    : ST_MAGAZINE_DIAG; // Состояние автомата магазина
	Error   : ST_MAGAZINE_ERRORS; // Активные и последние ошибки
END_VAR
VAR_IN_OUT
	stDetail : ARRAY [1..GVL_CELL_SETTINGS.NumberDetail] OF ST_DETAIL; // Содержимое слотов магазина
	stPoint  : ARRAY [0..GVL_POINT.iPointNumber] OF ST_POINT; // Глобальная таблица точек робота
END_VAR
VAR
	eGrantedOperation : E_MAGAZINE_OPERATION; // Доступная операция магазина
	eActualOperation  : E_MAGAZINE_OPERATION; // Выполняемая операция магазина

	rtExecute          : R_TRIG; // Фронт команды запуска
	rtEnable           : R_TRIG; // Фронт команды включения
	rtDisable          : R_TRIG; // Фронт команды отключения
	rtFillBlanks       : R_TRIG; // Фронт заполнения магазина заготовками
	rtClear            : R_TRIG; // Фронт очистки магазина
	rtCycleSlot        : R_TRIG; // Фронт изменения выбранного слота

	xExecuteRequest    : BOOL; // Активный запрос выполнения операции
	xResetRequest      : BOOL; // Активный запрос сброса
	xStopRequest       : BOOL; // Активный запрос остановки
	xManualCommand     : BOOL; // Команда получена из ручного интерфейса
	xDisableRequest    : BOOL; // Сохранённый запрос отключения после текущей операции

	iActiveSlotCount   : SINT; // Число активных слотов выбранной матрицы
	iInventoryIndex    : SINT; // Индекс изменения содержимого магазина
	iTakeSlot          : SINT; // Слот выбранной заготовки
	iPutSlot           : SINT; // Выбранный свободный слот
	uiStep             : UINT; // Шаг последовательности робота
	uiIndex            : UINT; // Индекс слота для расчёта координат
	uiRow              : UINT; // Строка выбранного слота
	uiColumn           : UINT; // Столбец выбранного слота

	stTakePoint          : ST_POINT; // Рассчитанная рабочая точка взятия
	stPutPoint           : ST_POINT; // Рассчитанная рабочая точка укладки
	stActiveRobotCommand : ST_ROBOT_COMMAND; // Команда роботу текущего шага
	xFinishedCondition   : BOOL; // Текущее содержимое не позволяет продолжить цикл
END_VAR
VAR CONSTANT
	ERR_WRONG_OPERATION : DWORD := DWORD#16#0000_0001; // Недопустимая операция магазина
	ERR_NO_BLANK        : DWORD := DWORD#16#0000_0002; // В магазине нет заготовки
	ERR_NO_FREE_SLOT    : DWORD := DWORD#16#0000_0004; // В магазине нет свободного слота
	ERR_INVALID_SLOT    : DWORD := DWORD#16#0000_0008; // Недопустимый номер слота
	ERR_SLOT_CONTENT    : DWORD := DWORD#16#0000_0010; // Содержимое слота не соответствует операции
	ERR_ROBOT           : DWORD := DWORD#16#0000_0020; // Ошибка робота при операции магазина
	ERR_GLOBAL_STOP     : DWORD := DWORD#16#0000_0040; // Остановка по глобальной ошибке
	ERR_GEOMETRY        : DWORD := DWORD#16#0000_0080; // Ошибка параметров матрицы магазина
	MASK_LOCAL_ERROR    : DWORD := ERR_WRONG_OPERATION OR ERR_NO_BLANK OR ERR_NO_FREE_SLOT
		OR ERR_INVALID_SLOT OR ERR_SLOT_CONTENT OR ERR_GEOMETRY; // Собственные первопричины магазина
END_VAR

// --- BEGIN IMPLEMENTATION ---

rtFillBlanks(CLK := xHmiFillBlanks);
rtClear(CLK := xHmiClear);
rtCycleSlot(CLK := xHmiCycleSlot);

// Активный размер матрицы может быть меньше полного массива деталей.
IF (uiRows > 0)
AND (uiColumns > 0)
AND ((uiRows * uiColumns) <= SINT_TO_UINT(GVL_CELL_SETTINGS.NumberDetail)) THEN
	iActiveSlotCount := UINT_TO_SINT(uiRows * uiColumns);
ELSE
	iActiveSlotCount := 0;
END_IF;

// Содержимое магазина изменяется только в отключенном состоянии.
IF Diag.eState = E_MAGAZINE_STATE.DISABLED THEN
	IF rtClear.Q THEN
		FOR iInventoryIndex := 1 TO GVL_CELL_SETTINGS.NumberDetail DO
			stDetail[iInventoryIndex].xInPosition := FALSE;
			stDetail[iInventoryIndex].eDetailType := E_DETAIL_TYPE.NONE;
		END_FOR;
	ELSIF rtFillBlanks.Q
	AND (iActiveSlotCount > 0) THEN
		FOR iInventoryIndex := 1 TO GVL_CELL_SETTINGS.NumberDetail DO
			stDetail[iInventoryIndex].xInPosition := iInventoryIndex <= iActiveSlotCount;
			IF iInventoryIndex <= iActiveSlotCount THEN
				stDetail[iInventoryIndex].eDetailType := E_DETAIL_TYPE.BLANK;
			ELSE
				stDetail[iInventoryIndex].eDetailType := E_DETAIL_TYPE.NONE;
			END_IF;
		END_FOR;
	ELSIF rtCycleSlot.Q
	AND (uiHmiEditSlot >= 1)
	AND (uiHmiEditSlot <= SINT_TO_UINT(iActiveSlotCount)) THEN
		iInventoryIndex := UINT_TO_SINT(uiHmiEditSlot);
		IF NOT stDetail[iInventoryIndex].xInPosition
		OR (stDetail[iInventoryIndex].eDetailType = E_DETAIL_TYPE.NONE) THEN
			stDetail[iInventoryIndex].xInPosition := TRUE;
			stDetail[iInventoryIndex].eDetailType := E_DETAIL_TYPE.BLANK;
		ELSIF stDetail[iInventoryIndex].eDetailType = E_DETAIL_TYPE.BLANK THEN
			stDetail[iInventoryIndex].xInPosition := TRUE;
			stDetail[iInventoryIndex].eDetailType := E_DETAIL_TYPE.DETAIL;
		ELSE
			stDetail[iInventoryIndex].xInPosition := FALSE;
			stDetail[iInventoryIndex].eDetailType := E_DETAIL_TYPE.NONE;
		END_IF;
	END_IF;
END_IF;

IF iActiveSlotCount > 0 THEN
	Status.iCurrentBlank := FindBlank(
		stDetail := stDetail,
		iSlotCount := iActiveSlotCount
	);
	Status.iCurrentFreeSlot := FindFreeSlot(
		stDetail := stDetail,
		iSlotCount := iActiveSlotCount
	);
ELSE
	Status.iCurrentBlank := 0;
	Status.iCurrentFreeSlot := 0;
END_IF;

Status.xOutBlank := Status.iCurrentBlank = 0;
Status.xOutFreeSlot := Status.iCurrentFreeSlot = 0;
Status.xCanTake := NOT Status.xOutBlank;
Status.xCanPut := NOT Status.xOutFreeSlot;
Status.xCanChange := Status.xCanTake AND Status.xCanPut;
Status.xCanEnable := FALSE;

IF stRobotStatus.xBlankAvailable
AND NOT stRobotStatus.xDetailAvailable THEN
	Status.xCanEnable := Status.xCanPut;
ELSIF stRobotStatus.xDetailAvailable
AND NOT stRobotStatus.xBlankAvailable THEN
	Status.xCanEnable := Status.xCanPut;
ELSIF NOT stRobotStatus.xBlankAvailable
AND NOT stRobotStatus.xDetailAvailable THEN
	Status.xCanEnable := Status.xCanTake;
END_IF;

xFinishedCondition :=
	(NOT stRobotStatus.xBlankAvailable
		AND NOT stRobotStatus.xDetailAvailable
		AND NOT Status.xCanTake)
	OR (stRobotStatus.xBlankAvailable
		AND NOT stRobotStatus.xDetailAvailable
		AND NOT Status.xCanPut)
	OR (NOT stRobotStatus.xBlankAvailable
		AND stRobotStatus.xDetailAvailable
		AND NOT Status.xCanPut);

// Автоматический выбор доступной операции.
eGrantedOperation := E_MAGAZINE_OPERATION.NONE;

IF NOT Status.xOutBlank
AND NOT stRobotStatus.xBlankAvailable
AND NOT stRobotStatus.xDetailAvailable THEN
	eGrantedOperation := E_MAGAZINE_OPERATION.TAKE;

ELSIF NOT Status.xOutFreeSlot
AND Status.xOutBlank
AND stRobotStatus.xDetailAvailable THEN
	eGrantedOperation := E_MAGAZINE_OPERATION.PUT;

ELSIF NOT Status.xOutFreeSlot
AND NOT Status.xOutBlank
AND stRobotStatus.xDetailAvailable THEN
	eGrantedOperation := E_MAGAZINE_OPERATION.CHANGE;
END_IF;

// Команды магазина с HMI принимаются только в ручном режиме.
xManualCommand := xManual AND (
	(stHmiCommand.eSetPoint = E_POINT_NAME.MAGAZINE_TAKE_DETAIL)
	OR (stHmiCommand.eSetPoint = E_POINT_NAME.MAGAZINE_PUT_DETAIL)
	OR (stHmiCommand.eSetPoint = E_POINT_NAME.MAGAZINE_CHANGE_DETAIL)
);

IF xManual THEN
	IF xManualCommand THEN
		xExecuteRequest := stHmiCommand.xExecute;
		xStopRequest := stHmiCommand.xStop;
	ELSE
		xExecuteRequest := FALSE;
		xStopRequest := FALSE;
	END_IF;
ELSE
	xExecuteRequest := stMagazineCommand.xExecute;
	xStopRequest := stMagazineCommand.xStop;
END_IF;

xResetRequest := xReset;

rtEnable(CLK := xHmiEnable OR (NOT xManual AND stMagazineCommand.xEnable));
rtDisable(CLK := xHmiDisable OR (NOT xManual AND stMagazineCommand.xDisable));

IF rtDisable.Q THEN
	xDisableRequest := TRUE;
END_IF;

rtExecute(CLK := xExecuteRequest);

// Значения команды роботу по умолчанию.
Command.xExecute := FALSE;
Command.xStop := FALSE;
Command.xReset := xResetRequest;
Command.eAction := E_ROBOT_ACTION.NONE;
Command.eSetPoint := E_POINT_NAME.NONE;
Command.iTakeSlot := 0;
Command.iPutSlot := 0;

IF xGlobalError
AND (Diag.eState <> E_MAGAZINE_STATE.DISABLED)
AND (Diag.eState <> E_MAGAZINE_STATE.IDLE)
AND (Diag.eState <> E_MAGAZINE_STATE.ERROR) THEN
	Error.dwErrorActive := Error.dwErrorActive OR ERR_GLOBAL_STOP;
	Diag.eState := E_MAGAZINE_STATE.ERROR;
END_IF;

CASE Diag.eState OF
	E_MAGAZINE_STATE.DISABLED:
		xDisableRequest := FALSE;
		IF rtEnable.Q
		AND Status.xCanEnable
		AND NOT xGlobalError THEN
			Diag.eState := E_MAGAZINE_STATE.IDLE;
		END_IF;

	E_MAGAZINE_STATE.IDLE:
		uiStep := 0;
		eActualOperation := E_MAGAZINE_OPERATION.NONE;

		IF xFinishedCondition THEN
			Diag.eState := E_MAGAZINE_STATE.DISABLED;
		ELSIF xDisableRequest THEN
			Diag.eState := E_MAGAZINE_STATE.DISABLED;
		ELSIF xGlobalError THEN
			Error.dwErrorActive := Error.dwErrorActive OR ERR_GLOBAL_STOP;
			Diag.eState := E_MAGAZINE_STATE.ERROR;
		ELSIF rtExecute.Q THEN
			IF xManualCommand THEN
				CASE stHmiCommand.eSetPoint OF
					E_POINT_NAME.MAGAZINE_TAKE_DETAIL:
						eActualOperation := E_MAGAZINE_OPERATION.TAKE;
					E_POINT_NAME.MAGAZINE_PUT_DETAIL:
						eActualOperation := E_MAGAZINE_OPERATION.PUT;
					E_POINT_NAME.MAGAZINE_CHANGE_DETAIL:
						eActualOperation := E_MAGAZINE_OPERATION.CHANGE;
				ELSE
					eActualOperation := E_MAGAZINE_OPERATION.NONE;
				END_CASE;
				iTakeSlot := stHmiCommand.iTakeSlot;
				iPutSlot := stHmiCommand.iPutSlot;
			ELSE
				eActualOperation := eGrantedOperation;
				iTakeSlot := Status.iCurrentBlank;
				iPutSlot := Status.iCurrentFreeSlot;
			END_IF;

			Diag.eState := E_MAGAZINE_STATE.CHOOSE;
		END_IF;

	E_MAGAZINE_STATE.CHOOSE:
		IF (iActiveSlotCount = 0)
		OR (NOT xMode AND (
			((uiColumns > 1) AND (lrPitchX = 0.0))
			OR ((uiRows > 1) AND (lrPitchY = 0.0))
			OR (lrSafeZ_1 = stPoint[E_POINT_NAME.MAGAZINE_DETAIL].Z)
			OR (stPoint[E_POINT_NAME.MAGAZINE_DETAIL].SpeedFactor <= 0.1)
			OR (stPoint[E_POINT_NAME.MAGAZINE_DETAIL].SpeedFactor > 1.0)
		)) THEN
			Error.dwErrorActive := Error.dwErrorActive OR ERR_GEOMETRY;
			Diag.eState := E_MAGAZINE_STATE.ERROR;

		ELSIF eActualOperation = E_MAGAZINE_OPERATION.NONE THEN
			Error.dwErrorActive := Error.dwErrorActive OR ERR_WRONG_OPERATION;
			Diag.eState := E_MAGAZINE_STATE.ERROR;

		ELSIF ((eActualOperation = E_MAGAZINE_OPERATION.TAKE)
			OR (eActualOperation = E_MAGAZINE_OPERATION.CHANGE))
		AND ((iTakeSlot < 1) OR (iTakeSlot > iActiveSlotCount)) THEN
			Error.dwErrorActive := Error.dwErrorActive OR ERR_NO_BLANK OR ERR_INVALID_SLOT;
			Diag.eState := E_MAGAZINE_STATE.ERROR;

		ELSIF ((eActualOperation = E_MAGAZINE_OPERATION.PUT)
			OR (eActualOperation = E_MAGAZINE_OPERATION.CHANGE))
		AND ((iPutSlot < 1) OR (iPutSlot > iActiveSlotCount)) THEN
			Error.dwErrorActive := Error.dwErrorActive OR ERR_NO_FREE_SLOT OR ERR_INVALID_SLOT;
			Diag.eState := E_MAGAZINE_STATE.ERROR;

		ELSIF ((eActualOperation = E_MAGAZINE_OPERATION.TAKE)
			OR (eActualOperation = E_MAGAZINE_OPERATION.CHANGE))
		AND (NOT stDetail[iTakeSlot].xInPosition
			OR (stDetail[iTakeSlot].eDetailType <> E_DETAIL_TYPE.BLANK)) THEN
			Error.dwErrorActive := Error.dwErrorActive OR ERR_SLOT_CONTENT;
			Diag.eState := E_MAGAZINE_STATE.ERROR;

		ELSIF ((eActualOperation = E_MAGAZINE_OPERATION.PUT)
			OR (eActualOperation = E_MAGAZINE_OPERATION.CHANGE))
		AND stDetail[iPutSlot].xInPosition THEN
			Error.dwErrorActive := Error.dwErrorActive OR ERR_SLOT_CONTENT;
			Diag.eState := E_MAGAZINE_STATE.ERROR;

		ELSIF (eActualOperation = E_MAGAZINE_OPERATION.TAKE)
		AND (stRobotStatus.xBlankAvailable OR stRobotStatus.xDetailAvailable) THEN
			Error.dwErrorActive := Error.dwErrorActive OR ERR_WRONG_OPERATION;
			Diag.eState := E_MAGAZINE_STATE.ERROR;

		ELSIF ((eActualOperation = E_MAGAZINE_OPERATION.PUT)
			OR (eActualOperation = E_MAGAZINE_OPERATION.CHANGE))
		AND NOT stRobotStatus.xDetailAvailable THEN
			Error.dwErrorActive := Error.dwErrorActive OR ERR_WRONG_OPERATION;
			Diag.eState := E_MAGAZINE_STATE.ERROR;

		ELSE
			IF (eActualOperation = E_MAGAZINE_OPERATION.TAKE)
			OR (eActualOperation = E_MAGAZINE_OPERATION.CHANGE) THEN
				uiIndex := SINT_TO_UINT(iTakeSlot - 1);
				uiColumn := uiIndex MOD uiColumns;
				uiRow := uiIndex / uiColumns;
				stTakePoint := stPoint[E_POINT_NAME.MAGAZINE_DETAIL];
				stTakePoint.X := stTakePoint.X + UINT_TO_LREAL(uiColumn) * lrPitchX;
				stTakePoint.Y := stTakePoint.Y + UINT_TO_LREAL(uiRow) * lrPitchY;
			END_IF;

			IF (eActualOperation = E_MAGAZINE_OPERATION.PUT)
			OR (eActualOperation = E_MAGAZINE_OPERATION.CHANGE) THEN
				uiIndex := SINT_TO_UINT(iPutSlot - 1);
				uiColumn := uiIndex MOD uiColumns;
				uiRow := uiIndex / uiColumns;
				stPutPoint := stPoint[E_POINT_NAME.MAGAZINE_DETAIL];
				stPutPoint.X := stPutPoint.X + UINT_TO_LREAL(uiColumn) * lrPitchX;
				stPutPoint.Y := stPutPoint.Y + UINT_TO_LREAL(uiRow) * lrPitchY;
			END_IF;

			uiStep := 0;
			Diag.eState := E_MAGAZINE_STATE.PREPARE_STEP;
		END_IF;

	E_MAGAZINE_STATE.PREPARE_STEP:
		stActiveRobotCommand.xExecute := FALSE;
		stActiveRobotCommand.xStop := FALSE;
		stActiveRobotCommand.xReset := xResetRequest;
		stActiveRobotCommand.eAction := E_ROBOT_ACTION.NONE;
		stActiveRobotCommand.eSetPoint := E_POINT_NAME.NONE;
		stActiveRobotCommand.iTakeSlot := iTakeSlot;
		stActiveRobotCommand.iPutSlot := iPutSlot;

		IF xMode THEN
			stActiveRobotCommand.eAction := E_ROBOT_ACTION.MOVE_TO_POINT;
			CASE eActualOperation OF
				E_MAGAZINE_OPERATION.TAKE:
					stActiveRobotCommand.eSetPoint := E_POINT_NAME.MAGAZINE_TAKE_DETAIL;
				E_MAGAZINE_OPERATION.PUT:
					stActiveRobotCommand.eSetPoint := E_POINT_NAME.MAGAZINE_PUT_DETAIL;
				E_MAGAZINE_OPERATION.CHANGE:
					stActiveRobotCommand.eSetPoint := E_POINT_NAME.MAGAZINE_CHANGE_DETAIL;
			END_CASE;
			Diag.eState := E_MAGAZINE_STATE.ROBOT_COMMAND;

		ELSE
			CASE eActualOperation OF
				E_MAGAZINE_OPERATION.TAKE:
					CASE uiStep OF
						0:
							IF stRobotStatus.xRotatedToDetail THEN
								Diag.eState := E_MAGAZINE_STATE.NEXT;
							ELSE
								stActiveRobotCommand.eAction := E_ROBOT_ACTION.ROTATE_TO_DETAIL;
							END_IF;
						1:
							stPoint[E_POINT_NAME.MAGAZINE_TAKE_DETAIL] := stTakePoint;
							stPoint[E_POINT_NAME.MAGAZINE_TAKE_DETAIL].Z := lrSafeZ_1;
							stActiveRobotCommand.eAction := E_ROBOT_ACTION.MOVE_TO_POINT;
							stActiveRobotCommand.eSetPoint := E_POINT_NAME.MAGAZINE_TAKE_DETAIL;
						2:
							stPoint[E_POINT_NAME.MAGAZINE_TAKE_DETAIL] := stTakePoint;
							stActiveRobotCommand.eAction := E_ROBOT_ACTION.MOVE_TO_POINT;
							stActiveRobotCommand.eSetPoint := E_POINT_NAME.MAGAZINE_TAKE_DETAIL;
						3: stActiveRobotCommand.eAction := E_ROBOT_ACTION.CLAMP_1;
						4:
							stPoint[E_POINT_NAME.MAGAZINE_TAKE_DETAIL] := stTakePoint;
							stPoint[E_POINT_NAME.MAGAZINE_TAKE_DETAIL].Z := lrSafeZ_1;
							stActiveRobotCommand.eAction := E_ROBOT_ACTION.MOVE_TO_POINT;
							stActiveRobotCommand.eSetPoint := E_POINT_NAME.MAGAZINE_TAKE_DETAIL;
					ELSE
						Diag.eState := E_MAGAZINE_STATE.DONE;
					END_CASE;

				E_MAGAZINE_OPERATION.PUT:
					CASE uiStep OF
						0:
							IF stRobotStatus.xRotatedToBlank THEN
								Diag.eState := E_MAGAZINE_STATE.NEXT;
							ELSE
								stActiveRobotCommand.eAction := E_ROBOT_ACTION.ROTATE_TO_BLANK;
							END_IF;
						1:
							stPoint[E_POINT_NAME.MAGAZINE_PUT_DETAIL] := stPutPoint;
							stPoint[E_POINT_NAME.MAGAZINE_PUT_DETAIL].Z := lrSafeZ_1;
							stActiveRobotCommand.eAction := E_ROBOT_ACTION.MOVE_TO_POINT;
							stActiveRobotCommand.eSetPoint := E_POINT_NAME.MAGAZINE_PUT_DETAIL;
						2:
							stPoint[E_POINT_NAME.MAGAZINE_PUT_DETAIL] := stPutPoint;
							stActiveRobotCommand.eAction := E_ROBOT_ACTION.MOVE_TO_POINT;
							stActiveRobotCommand.eSetPoint := E_POINT_NAME.MAGAZINE_PUT_DETAIL;
						3: stActiveRobotCommand.eAction := E_ROBOT_ACTION.UNCLAMP_2;
						4:
							stPoint[E_POINT_NAME.MAGAZINE_PUT_DETAIL] := stPutPoint;
							stPoint[E_POINT_NAME.MAGAZINE_PUT_DETAIL].Z := lrSafeZ_1;
							stActiveRobotCommand.eAction := E_ROBOT_ACTION.MOVE_TO_POINT;
							stActiveRobotCommand.eSetPoint := E_POINT_NAME.MAGAZINE_PUT_DETAIL;
					ELSE
						Diag.eState := E_MAGAZINE_STATE.DONE;
					END_CASE;

				E_MAGAZINE_OPERATION.CHANGE:
					CASE uiStep OF
						0:
							IF stRobotStatus.xRotatedToBlank THEN
								Diag.eState := E_MAGAZINE_STATE.NEXT;
							ELSE
								stActiveRobotCommand.eAction := E_ROBOT_ACTION.ROTATE_TO_BLANK;
							END_IF;
						1:
							stPoint[E_POINT_NAME.MAGAZINE_PUT_DETAIL] := stPutPoint;
							stPoint[E_POINT_NAME.MAGAZINE_PUT_DETAIL].Z := lrSafeZ_1;
							stActiveRobotCommand.eAction := E_ROBOT_ACTION.MOVE_TO_POINT;
							stActiveRobotCommand.eSetPoint := E_POINT_NAME.MAGAZINE_PUT_DETAIL;
						2:
							stPoint[E_POINT_NAME.MAGAZINE_PUT_DETAIL] := stPutPoint;
							stActiveRobotCommand.eAction := E_ROBOT_ACTION.MOVE_TO_POINT;
							stActiveRobotCommand.eSetPoint := E_POINT_NAME.MAGAZINE_PUT_DETAIL;
						3: stActiveRobotCommand.eAction := E_ROBOT_ACTION.UNCLAMP_2;
						4:
							stPoint[E_POINT_NAME.MAGAZINE_PUT_DETAIL] := stPutPoint;
							stPoint[E_POINT_NAME.MAGAZINE_PUT_DETAIL].Z := lrSafeZ_2;
							stActiveRobotCommand.eAction := E_ROBOT_ACTION.MOVE_TO_POINT;
							stActiveRobotCommand.eSetPoint := E_POINT_NAME.MAGAZINE_PUT_DETAIL;
						5:
							IF stRobotStatus.xRotatedToDetail THEN
								Diag.eState := E_MAGAZINE_STATE.NEXT;
							ELSE
								stActiveRobotCommand.eAction := E_ROBOT_ACTION.ROTATE_TO_DETAIL;
							END_IF;
						6:
							stPoint[E_POINT_NAME.MAGAZINE_TAKE_DETAIL] := stTakePoint;
							stPoint[E_POINT_NAME.MAGAZINE_TAKE_DETAIL].Z := lrSafeZ_2;
							stActiveRobotCommand.eAction := E_ROBOT_ACTION.MOVE_TO_POINT;
							stActiveRobotCommand.eSetPoint := E_POINT_NAME.MAGAZINE_TAKE_DETAIL;
						7:
							stPoint[E_POINT_NAME.MAGAZINE_TAKE_DETAIL] := stTakePoint;
							stActiveRobotCommand.eAction := E_ROBOT_ACTION.MOVE_TO_POINT;
							stActiveRobotCommand.eSetPoint := E_POINT_NAME.MAGAZINE_TAKE_DETAIL;
						8: stActiveRobotCommand.eAction := E_ROBOT_ACTION.CLAMP_1;
						9:
							stPoint[E_POINT_NAME.MAGAZINE_TAKE_DETAIL] := stTakePoint;
							stPoint[E_POINT_NAME.MAGAZINE_TAKE_DETAIL].Z := lrSafeZ_1;
							stActiveRobotCommand.eAction := E_ROBOT_ACTION.MOVE_TO_POINT;
							stActiveRobotCommand.eSetPoint := E_POINT_NAME.MAGAZINE_TAKE_DETAIL;
					ELSE
						Diag.eState := E_MAGAZINE_STATE.DONE;
					END_CASE;
			END_CASE;

			IF Diag.eState = E_MAGAZINE_STATE.PREPARE_STEP THEN
				Diag.eState := E_MAGAZINE_STATE.ROBOT_COMMAND;
			END_IF;
		END_IF;

	E_MAGAZINE_STATE.ROBOT_COMMAND:
		Command := stActiveRobotCommand;
		Command.xExecute := TRUE;

		IF xStopRequest OR xGlobalError THEN
			Command.xStop := TRUE;
			Error.dwErrorActive := Error.dwErrorActive OR ERR_GLOBAL_STOP;
			Diag.eState := E_MAGAZINE_STATE.ERROR;

		ELSIF stRobotStatus.xError THEN
			Error.dwErrorActive := Error.dwErrorActive OR ERR_ROBOT;
			Diag.eState := E_MAGAZINE_STATE.ERROR;

		ELSIF stRobotStatus.xDone THEN
			IF xMode THEN
				IF (eActualOperation = E_MAGAZINE_OPERATION.PUT)
				OR (eActualOperation = E_MAGAZINE_OPERATION.CHANGE) THEN
					stDetail[iPutSlot].xInPosition := TRUE;
					stDetail[iPutSlot].eDetailType := E_DETAIL_TYPE.DETAIL;
				END_IF;
				IF (eActualOperation = E_MAGAZINE_OPERATION.TAKE)
				OR (eActualOperation = E_MAGAZINE_OPERATION.CHANGE) THEN
					stDetail[iTakeSlot].xInPosition := FALSE;
					stDetail[iTakeSlot].eDetailType := E_DETAIL_TYPE.NONE;
				END_IF;
			ELSE
				IF (uiStep = 3)
				AND ((eActualOperation = E_MAGAZINE_OPERATION.PUT)
					OR (eActualOperation = E_MAGAZINE_OPERATION.CHANGE)) THEN
					stDetail[iPutSlot].xInPosition := TRUE;
					stDetail[iPutSlot].eDetailType := E_DETAIL_TYPE.DETAIL;
				END_IF;
				IF ((uiStep = 3) AND (eActualOperation = E_MAGAZINE_OPERATION.TAKE))
				OR ((uiStep = 8) AND (eActualOperation = E_MAGAZINE_OPERATION.CHANGE)) THEN
					stDetail[iTakeSlot].xInPosition := FALSE;
					stDetail[iTakeSlot].eDetailType := E_DETAIL_TYPE.NONE;
				END_IF;
			END_IF;

			Diag.eState := E_MAGAZINE_STATE.RELEASE_ROBOT_COMMAND;
		END_IF;

	E_MAGAZINE_STATE.RELEASE_ROBOT_COMMAND:
		IF stRobotStatus.xError THEN
			Error.dwErrorActive := Error.dwErrorActive OR ERR_ROBOT;
			Diag.eState := E_MAGAZINE_STATE.ERROR;
		ELSIF NOT stRobotStatus.xBusy AND NOT stRobotStatus.xDone THEN
			IF xMode THEN
				Diag.eState := E_MAGAZINE_STATE.DONE;
			ELSE
				Diag.eState := E_MAGAZINE_STATE.NEXT;
			END_IF;
		END_IF;

	E_MAGAZINE_STATE.NEXT:
		uiStep := uiStep + 1;
		Diag.eState := E_MAGAZINE_STATE.PREPARE_STEP;

	E_MAGAZINE_STATE.DONE:
		IF NOT xExecuteRequest THEN
			eActualOperation := E_MAGAZINE_OPERATION.NONE;
			IF xDisableRequest THEN
				Diag.eState := E_MAGAZINE_STATE.DISABLED;
			ELSE
				Diag.eState := E_MAGAZINE_STATE.IDLE;
			END_IF;
		END_IF;

	E_MAGAZINE_STATE.ERROR:
		IF stRobotStatus.xBusy THEN
			Command := stActiveRobotCommand;
			Command.xExecute := TRUE;
			Command.xStop := TRUE;
		END_IF;

		IF xResetRequest
		AND NOT xExecuteRequest
		AND NOT xGlobalError
		AND NOT stRobotStatus.xError THEN
			Error.dwErrorLast := Error.dwErrorActive;
			Error.dwErrorActive := DWORD#0;
			eActualOperation := E_MAGAZINE_OPERATION.NONE;
			Diag.eState := E_MAGAZINE_STATE.DISABLED;
		END_IF;
END_CASE;

Status.xEnabled := Diag.eState <> E_MAGAZINE_STATE.DISABLED;
Status.xDisablePending := xDisableRequest AND Status.xEnabled;
Status.xReady := Diag.eState = E_MAGAZINE_STATE.IDLE;
Status.xBusy := (Diag.eState <> E_MAGAZINE_STATE.DISABLED)
	AND (Diag.eState <> E_MAGAZINE_STATE.IDLE)
	AND (Diag.eState <> E_MAGAZINE_STATE.DONE)
	AND (Diag.eState <> E_MAGAZINE_STATE.ERROR);
Status.xDone := Diag.eState = E_MAGAZINE_STATE.DONE;
Status.xError := Diag.eState = E_MAGAZINE_STATE.ERROR;
Status.eGrantedOperation := eGrantedOperation;
Status.eActualOperation := eActualOperation;
Status.iSelectedBlank := iTakeSlot;
Status.iSelectedFreeSlot := iPutSlot;
Status.xFinished := xFinishedCondition AND NOT Status.xBusy;
Error.dwAlarmActive := Error.dwErrorActive AND MASK_LOCAL_ERROR;

IF Error.dwErrorActive <> DWORD#0 THEN
	Error.dwErrorLast := Error.dwErrorActive;
END_IF;

Error.stErrorActive := UpdateErrorView(dwError := Error.dwErrorActive);
Error.stErrorLast := UpdateErrorView(dwError := Error.dwErrorLast);

(* ---- FB_MOTION_MANAGER.st ---- *)
FUNCTION_BLOCK FB_MOTION_MANAGER
VAR_INPUT
	stPoint : ARRAY [0..GVL_POINT.iPointNumber] OF ST_POINT; // Глобальная таблица точек
	xReset  : BOOL; // Сброс ошибок менеджера движения
END_VAR
VAR_OUTPUT
END_VAR
VAR
	curPoint      : ST_POINT; // Координаты выбранной точки
	curPointName  : E_POINT_NAME; // Имя выбранной точки
	fbPointManager: FB_POINT_MANAGER; // Проверка координат и скорости точки
END_VAR
VAR CONSTANT
	ERR_POINT_INVALID : DWORD := DWORD#16#0000_0001; // Недопустимая точка
	ERR_GROUP         : DWORD := DWORD#16#0000_0002; // Ошибка группы осей
	ERR_GLOBAL_STOP   : DWORD := DWORD#16#0000_0004; // Глобальная ошибка ячейки
END_VAR
VAR_IN_OUT
	stMotionManager : ST_MOTION_MANAGER; // Команды, статусы и диагностика менеджера движения
	GroupData       : ST_AXIS_GROUP; // Команды, статусы и диагностика группы XYZ
	stPointManager  : ST_POINT_MANAGER; // Команды, статусы и диагностика проверки точки
END_VAR

// --- BEGIN IMPLEMENTATION ---

stPointManager.Diag.lrX_MinLimit := -1000;
stPointManager.Diag.lrX_MaxLimit := 17000;
stPointManager.Diag.lrY_MinLimit := -1000;
stPointManager.Diag.lrY_MaxLimit := 17000;
stPointManager.Diag.lrZ_MinLimit := -1000;
stPointManager.Diag.lrZ_MaxLimit := 17000;
fbPointManager(
			stPointManager := stPointManager,
			stPoint := curPoint
		);

stMotionManager.Status.xBusy := FALSE;
stMotionManager.Status.xDone := FALSE;
stMotionManager.Status.xError := FALSE;
stMotionManager.Status.xReady:= FALSE;
stMotionManager.Command.xReset := xReset;

CASE stMotionManager.Diag.eState OF
	// --------------------------------------------------
	E_MOTION_MANAGER_STATE.IDLE:
	// --------------------------------------------------
		stMotionManager.Status.xReady:= TRUE;
		IF stMotionManager.Command.xExecute AND NOT stMotionManager.Command.xGlobalError THEN
			stMotionManager.Status.xBusy := TRUE;
			stMotionManager.Diag.eState := E_MOTION_MANAGER_STATE.VALIDATE;
		ELSIF stMotionManager.Command.xGlobalError THEN
			stMotionManager.Error.dwErrorActive := stMotionManager.Error.dwErrorActive OR ERR_GLOBAL_STOP;
			stMotionManager.Diag.eState := E_MOTION_MANAGER_STATE.ERROR;
		END_IF

	// --------------------------------------------------
	E_MOTION_MANAGER_STATE.VALIDATE:
	// --------------------------------------------------
		stMotionManager.Status.xBusy := TRUE;
		curPoint := stPoint[stMotionManager.Command.eTargetPoint];
		curPointName := stMotionManager.Command.eTargetPoint;

		stPointManager.Command.xExecute := TRUE;

		IF stPointManager.Status.xDone AND NOT stPointManager.Status.xInvalid THEN
			stPointManager.Command.xExecute := FALSE;
			IF stMotionManager.Command.xMode THEN
				stMotionManager.Diag.eState := 	E_MOTION_MANAGER_STATE.MOTION_MODBUS;
			ELSE
				stMotionManager.Diag.eState := 	E_MOTION_MANAGER_STATE.MOTION_SIM;
			END_IF
		ELSIF stPointManager.Status.xDone AND stPointManager.Status.xInvalid THEN
			stMotionManager.Error.dwErrorActive := stMotionManager.Error.dwErrorActive OR ERR_POINT_INVALID;
			stMotionManager.Diag.eState := 	E_MOTION_MANAGER_STATE.ERROR;
		END_IF

	// --------------------------------------------------
	E_MOTION_MANAGER_STATE.MOTION_SIM:
	// --------------------------------------------------

		stMotionManager.Status.xBusy := TRUE;

		GroupData.MotionParam.lrX := curPoint.X;
		GroupData.MotionParam.lrY := curPoint.Y;
		GroupData.MotionParam.lrZ := curPoint.Z;
		GroupData.MotionParam.VelFactor := curPoint.SpeedFactor;
		GroupData.MotionParam.AccFactor := curPoint.SpeedFactor;
		GroupData.MotionParam.JerkFactor := curPoint.SpeedFactor;
		IF GroupData.Diag.iStep = E_AXIS_GROUP_STATE.READY AND NOT GroupData.Command.xMoveDirect AND NOT stMotionManager.Command.xGlobalError THEN
			GroupData.Command.xMoveDirect := TRUE;
		END_IF;

		IF GroupData.Status.xMoveDirectDone AND GroupData.Command.xMoveDirect THEN
			GroupData.Command.xMoveDirect := FALSE;
			stMotionManager.Status.eCurrentPoint := curPointName;
			stMotionManager.Diag.eState := 	E_MOTION_MANAGER_STATE.DONE;
		ELSIF GroupData.Diag.iStep = E_AXIS_GROUP_STATE.ERROR OR stMotionManager.Command.xGlobalError  THEN
			IF GroupData.Diag.iStep = E_AXIS_GROUP_STATE.ERROR THEN
				stMotionManager.Error.dwErrorActive := stMotionManager.Error.dwErrorActive OR ERR_GROUP;
			END_IF;
			IF stMotionManager.Command.xGlobalError THEN
				stMotionManager.Error.dwErrorActive := stMotionManager.Error.dwErrorActive OR ERR_GLOBAL_STOP;
			END_IF;
			stMotionManager.Diag.eState := 	E_MOTION_MANAGER_STATE.ERROR;
		END_IF

	// --------------------------------------------------
	E_MOTION_MANAGER_STATE.ERROR:
	// --------------------------------------------------
		stMotionManager.Status.xError := TRUE;
		IF NOT stMotionManager.Command.xGlobalError AND stMotionManager.Command.xReset THEN
			stMotionManager.Error.dwErrorLast := stMotionManager.Error.dwErrorActive;
			stMotionManager.Error.dwErrorActive := DWORD#0;
			stMotionManager.Status.xError := FALSE;
			stMotionManager.Diag.eState := 	E_MOTION_MANAGER_STATE.IDLE;
		END_IF

	// --------------------------------------------------
	E_MOTION_MANAGER_STATE.DONE:
	// --------------------------------------------------
		stMotionManager.Status.xBusy := FALSE;
		stMotionManager.Status.xDone := TRUE;
		IF NOT stMotionManager.Command.xExecute THEN
			stMotionManager.Diag.eState := 	E_MOTION_MANAGER_STATE.IDLE;
		END_IF
	END_CASE

// Все текущие ошибки менеджера являются следствием точки, группы или внешней остановки.
stMotionManager.Error.dwAlarmActive := DWORD#0;

stMotionManager.Error.stErrorActive := UpdateErrorView(
	dwError := stMotionManager.Error.dwErrorActive
);
stMotionManager.Error.stErrorLast := UpdateErrorView(
	dwError := stMotionManager.Error.dwErrorLast
);

(* ---- FB_POINT_MANAGER.st ---- *)
FUNCTION_BLOCK FB_POINT_MANAGER
VAR_INPUT
	stPoint : ST_POINT; // Проверяемая точка
END_VAR
VAR_OUTPUT
END_VAR
VAR
END_VAR
VAR_IN_OUT
	stPointManager : ST_POINT_MANAGER; // Команды, статусы и диагностика проверки точки
END_VAR
VAR CONSTANT
	X_OUT_OF_LIMIT : DWORD := 1; // Координата X вне допустимых границ
	Y_OUT_OF_LIMIT : DWORD := 2; // Координата Y вне допустимых границ
	Z_OUT_OF_LIMIT : DWORD := 4; // Координата Z вне допустимых границ
	INVALID_VEL    : DWORD := 8; // Недопустимый коэффициент скорости
END_VAR

// --- BEGIN IMPLEMENTATION ---

stPointManager.Status.xBusy := FALSE;
stPointManager.Status.xDone := FALSE;
stPointManager.Status.xInvalid := FALSE;

CASE stPointManager.Diag.eState OF
	// --------------------------------------------------
	E_POINT_MANAGER_STATE.IDLE:
	// --------------------------------------------------
		stPointManager.Error.dwErrorActive := DWORD#0;
		IF stPointManager.Command.xExecute THEN
			stPointManager.Status.xBusy := TRUE;
			stPointManager.Diag.eState := E_POINT_MANAGER_STATE.CHECK_ZONE;
		END_IF

	// --------------------------------------------------
	E_POINT_MANAGER_STATE.CHECK_ZONE:
	// --------------------------------------------------
		stPointManager.Status.xBusy := TRUE;

		IF NOT ((stPointManager.Diag.lrX_MinLimit <= stPoint.X) AND (stPoint.X <= stPointManager.Diag.lrX_MaxLimit)) THEN
			stPointManager.Error.dwErrorActive := stPointManager.Error.dwErrorActive OR X_OUT_OF_LIMIT;
		END_IF

		IF NOT ((stPointManager.Diag.lrY_MinLimit <= stPoint.Y) AND (stPoint.Y <= stPointManager.Diag.lrY_MaxLimit)) THEN
			stPointManager.Error.dwErrorActive := stPointManager.Error.dwErrorActive OR Y_OUT_OF_LIMIT;
		END_IF

		IF NOT ((stPointManager.Diag.lrZ_MinLimit <= stPoint.Z) AND (stPoint.Z <= stPointManager.Diag.lrZ_MaxLimit)) THEN
			stPointManager.Error.dwErrorActive := stPointManager.Error.dwErrorActive OR Z_OUT_OF_LIMIT;
		END_IF

		stPointManager.Diag.eState := E_POINT_MANAGER_STATE.CHECK_VEL_FACTOR;

	// --------------------------------------------------
	E_POINT_MANAGER_STATE.CHECK_VEL_FACTOR:
	// --------------------------------------------------
		stPointManager.Status.xBusy := TRUE;

		IF  NOT ((0.1 < stPoint.SpeedFactor) AND(stPoint.SpeedFactor <= 1.0))  THEN
			stPointManager.Error.dwErrorActive := stPointManager.Error.dwErrorActive OR INVALID_VEL;
		END_IF

		stPointManager.Diag.eState := E_POINT_MANAGER_STATE.CHECK_ALL;

	// --------------------------------------------------
	E_POINT_MANAGER_STATE.CHECK_ALL:
	// --------------------------------------------------
		stPointManager.Status.xDone := TRUE;
		stPointManager.Status.xBusy := FALSE;
		IF stPointManager.Error.dwErrorActive <> DWORD#0 THEN
			stPointManager.Status.xInvalid := TRUE;
			stPointManager.Error.dwErrorLast := stPointManager.Error.dwErrorActive;
		ELSE
			stPointManager.Status.xInvalid := FALSE;
		END_IF

		IF NOT stPointManager.Command.xExecute THEN
			stPointManager.Diag.eState := E_POINT_MANAGER_STATE.IDLE;
		END_IF

END_CASE

stPointManager.Error.dwAlarmActive := stPointManager.Error.dwErrorActive;

stPointManager.Error.stErrorActive := UpdateErrorView(
	dwError := stPointManager.Error.dwErrorActive
);
stPointManager.Error.stErrorLast := UpdateErrorView(
	dwError := stPointManager.Error.dwErrorLast
);
